METHOD PUBLIC closeAll : BOOL //Return value = TRUE if busy
VAR_INPUT
	Execute													:	BOOL;
END_VAR
	IF Execute
	THEN
		Error												:=	FALSE;
		ErrorId												:= 0;
		SocketCloseAll.bExecute 							:= TRUE;
	ELSIF NOT SocketCloseAll.bBusy  						
	THEN                            						
		Error												:= FALSE;
		ErrorId												:= 0;
		SocketCloseAll.bExecute 							:= FALSE;
	END_IF                          						
                                    	
	MemFnc													:= FNC_CLOSE_ALL;
	THIS^.Execute											:= Execute;

	SocketCloseAll(
		sSrvNetId	:= SrvNetId,
		bExecute	:= ,
		tTimeout	:= Timeout,
		bBusy		=> Busy,
		bError		=> ,
		nErrId		=> );

	IF NOT SocketCloseAll.bBusy
		AND NOT SocketCloseAll.bError
		AND SocketCloseAll.bExecute
	THEN
		Done												:= TRUE;
		MEMSET(ADR(hSocket), 0 , SIZEOF(hSocket));
		hSocketText											:= '';
		Online												:= FALSE;
	ELSE
		Done												:= FALSE;
	END_IF

	IF NOT Busy
	THEN
		IF SocketCloseAll.bExecute
		THEN
			Error											:=	SocketCloseAll.bError;
			IF SocketCloseAll.nErrId >= 16#80070000
			THEN
				ErrorId										:= E_AdsErr.CLIENT_W32ERROR;
				WinsockErrorId								:= ADSERROR_TO_WSERROR(SocketCloseAll.nErrId);
			ELSE                    						
				ErrorId										:= SocketCloseAll.nErrId;
				WinsockErrorId								:= WSOK;
			END_IF
		END_IF
		IF NOT Execute
		THEN
			MemFnc											:=  -1;
			SocketCloseAll(bExecute := FALSE);
		END_IF
	END_IF
	
	CloseAll												:= Busy;
END_METHOD

METHOD PUBLIC connect : BOOL //Return value = TRUE if busy
//required parameter
//Host
//Port
VAR_INPUT
	Execute													:	BOOL;	
END_VAR
	IF Execute
	THEN
		Error												:=	FALSE;
		ErrorId												:= 0;
		SocketCreate.bExecute 								:= TRUE;
	ELSIF NOT SocketCreate.bBusy    						
	THEN                            						
		Error												:=	FALSE;
		ErrorId												:= 0;
		SocketCreate.bExecute 								:= FALSE;
	END_IF                          						
                                    	
	MemFnc													:= FNC_CONNECT;
	THIS^.Execute											:= Execute;

	SocketCreate(
		sSrvNetId	:= SrvNetId,
		sRemoteHost	:= Host,
		nRemotePort	:= Port,
		bExecute	:= ,
		tTimeout	:= Timeout,
		bBusy		=> Busy,
		bError		=> ,
		nErrId		=> ,
		hSocket		=> );

	IF NOT SocketCreate.bBusy
		AND NOT SocketCreate.bError
		AND SocketCreate.bExecute
	THEN
		Done												:= TRUE;
		hSocket												:= SocketCreate.hSocket;
		hSocketText											:= HSOCKET_TO_STRING(hSocket);
		Online												:= SocketCreate.hSocket.handle <> 0;
	ELSE                                					
		Done												:= FALSE;
	END_IF                              	
                                        	
	IF NOT Busy
	THEN
		IF SocketCreate.bExecute
		THEN
			Error											:=	SocketCreate.bError;
			IF SocketCreate.nErrId >= 16#80070000
			THEN
				ErrorId										:= E_AdsErr.CLIENT_W32ERROR;
				WinsockErrorId								:= ADSERROR_TO_WSERROR(SocketCreate.nErrId);
			ELSE                    						
				ErrorId										:= SocketCreate.nErrId;
				WinsockErrorId								:= WSOK;
			END_IF                  						
		END_IF                      	
		IF NOT Execute              	
		THEN
			MemFnc											:= -1;
			SocketCreate(bExecute := FALSE);
		END_IF
	END_IF
	
	Connect													:= Busy;
END_METHOD

METHOD PUBLIC listen : BOOL //Return value = TRUE if busy
//required parameter
//hListener
//Host
//Port
VAR_INPUT
	Execute													:	BOOL;
END_VAR
	IF Execute
	THEN
		Error												:= FALSE;
		ErrorId												:= 0;
		SocketListen.bExecute 								:= TRUE;
	ELSIF NOT SocketListen.bBusy    						
	THEN                            						
		Error												:= FALSE;
		ErrorId												:= 0;
		SocketListen.bExecute 								:= FALSE;
	END_IF                          						
                                        					
	MemFnc													:= FNC_LISTEN;
	THIS^.Execute											:= Execute;
                                        	
	SocketListen(
		sSrvNetId	:= SrvNetId,
		sLocalHost	:= Host,
		nlocalPort	:= Port,
		bExecute	:= ,
		tTimeout	:= Timeout,
		bBusy		=> Busy,
		bError		=>,
		nErrId		=> ,
		hListener	=>	hSocket);

	IF NOT SocketListen.bBusy
		AND NOT SocketListen.bError
		AND SocketListen.bExecute
	THEN
		Done												:= TRUE;
		hSocket												:= SocketListen.hListener;
		hSocketText											:= HSOCKET_TO_STRING(hSocket);
		Request												:= TRUE;
	ELSE                            						
		Done												:= FALSE;
	END_IF                              					
                                        	
	IF NOT Busy
	THEN
		IF SocketListen.bExecute
		THEN
			Error											:=	SocketListen.bError;
			IF SocketListen.nErrId >= 16#80070000
			THEN
				ErrorId										:= E_AdsErr.CLIENT_W32ERROR;
				WinsockErrorId								:= ADSERROR_TO_WSERROR(SocketListen.nErrId);
			ELSE                    						
				ErrorId										:= SocketListen.nErrId;
				WinsockErrorId								:= WSOK;
			END_IF                  						
		END_IF                      	
		IF NOT Execute              	
		THEN                        	
			MemFnc											:= -1;
			SocketListen(bExecute := FALSE);
		END_IF
	END_IF
	
	Listen													:= Busy;
END_METHOD

END_FUNCTION_BLOCK

// POUs/Connectivity/TF6310-TcpServer/UDP/UDPSendRecCtrl
{attribute 'no_check'}
//Send or receive data via TCP connection 
//based on TF6310, required lib: Tc2_TcpIp - see Beckhoff Infosys for more information
FUNCTION_BLOCK UDPSendRecCtrl Extends FbBase
VAR_OUTPUT CONSTANT
	FNC_RECEIVE												:	INT := 0;
	FNC_SEND												:	INT := 1;
END_VAR             										
VAR_INPUT           										
	Fnc														:	INT (FNC_RECEIVE..FNC_SEND) := FNC_RECEIVE;
{attribute 'displaymode':='binary'}
	Options													:	BYTE := 2#0000_0000; // Options Bit .0 = Do NOT restart receive intern / Receive intern nicht neustarten
	SrvNetId												: 	T_AmsNetId := ''; 	// server ams net id
	RemoteHost 												: 	T_IPv4Addr; // Target ip adress - only for send data *)
	RemotePort												: 	UDINT; 	// target port - only for send data *)
	Timeout													: 	TIME := DEFAULT_ADS_TIMEOUT; //ADS timeout
	hSocket													:	T_HSOCKET; 	// Socket handle provided by Server/Handle
	pData													:	POINTER TO BYTE; 	//Pointer do send/res data field 
	cbData													:	UDINT; 	// Size of send/rec data field 
	EnableDebugMode											:	BOOL;	// Write debug information into twincat logger
END_VAR
VAR_OUTPUT
	RecBytes 												:  UDINT;  	// Count of received bytes
	WinsockErrorId											:	E_WinsockError; //Winsocket error enum - see TF6310 documentation for further information
	RecRemoteHost 											:  STRING(15); 	// Remote host IP
	RecRemotePort											:  UDINT; 	// Remote host port
END_VAR                 									
VAR                     	
(* cache ************************************************************)
	MemFnc													:	INT := -1;

(* function-block instances ***************************************************************)
	SocketSend												:	FB_SocketUdpSendTo;
	SocketReceive											:	FB_SocketUdpReceiveFrom;

END_VAR


(* Execute ***************************************************************************************)
	rtExecute(CLK := Execute);
	IF rtExecute.Q
		AND MemFnc < 0
	THEN
		MemFnc 												:= SEL(Fnc = FNC_SEND, FNC_RECEIVE , FNC_SEND) ;
		Busy												:= TRUE;
		Done												:= FALSE;
		Error												:= FALSE;
		ErrorID												:= 0;
	END_IF

(* Call Method ***********************************************************************************)
	CASE MemFnc OF
	FNC_SEND:
		SEND( Execute := Execute);

	FNC_RECEIVE:
		Receive( Execute := Execute);
			
	-1:
		IF NOT Execute
		THEN
			Busy											:= FALSE;
			Done											:= FALSE;
			Error											:= FALSE;
			ErrorID											:= 0;
		END_IF                              				
	ELSE                                    				
		Busy												:= FALSE;
		Done												:= FALSE;
		Error												:= Execute;
		ErrorID												:= E_AdsErr.DEVICE_INVALIDPARM;
	END_CASE                                	
                                            	
(*************************************************************************************************)

PROPERTY PUBLIC optDoNotRestartReceiveCylic : BOOL
GET
optDoNotRestartReceiveCylic := Options.0;
END_GET
SET
Options.0 := optDoNotRestartReceiveCylic;
END_SET
END_PROPERTY

METHOD PUBLIC receive : BOOL	//Return value = TRUE if busy
//required parameter
//hSocket
//pData
//cbData
VAR_INPUT
	Execute													:	BOOL;
END_VAR
	MemFnc													:= FNC_RECEIVE;
	THIS^.Execute											:= Execute;
	
IF pData = 0 
THEN
	Busy													:= NOT Error;
	Error													:= TRUE;
	ErrorId													:= E_AdsErr.DEVICE_INVALIDPARM;
	Done													:= FALSE;
	MemFnc													:= SEL(Execute , -1 ,MemFnc); 
	RETURN;
END_IF

	IF Execute
	THEN
		Error												:=	FALSE;
		ErrorId												:= 0;
		SocketReceive.bExecute 								:= TRUE;
	ELSIF NOT SocketReceive.bBusy       					
	THEN                                					
		Error												:=	FALSE;
		ErrorId												:= 0;
		SocketReceive.bExecute 								:= FALSE;
	END_IF

	SocketReceive(
		sSrvNetId	:= SrvNetId,
		hSocket		:= hSocket,
		cbLen		:= cbData,
		pDest		:= pData,
		bExecute	:= ,
		tTimeout	:= Timeout,
		bBusy		=> Busy,
		bError		=> ,
		nErrId		=> ,
		nRecBytes	=> );

	IF NOT SocketReceive.bBusy
		AND NOT SocketReceive.bError
		AND SocketReceive.bExecute
	THEN
		IF EnableDebugMode
			AND SocketReceive.nRecBytes > 0
			AND NOT Done
		THEN
			hSocket.remoteAddr.sAddr						:= SocketReceive.sRemoteHost;
			hSocket.remoteAddr.nPort						:= SocketReceive.nRemotePort;
			ADSLOGDINT(	ADSLOG_MSGTYPE_ERROR OR ADSLOG_MSGTYPE_LOG, CONCAT('%d Bytes received / ', HSOCKET_TO_STRING(hSocket)) , UDINT_TO_DINT(SocketReceive.nRecBytes));
		END_IF
		Done												:= SocketReceive.nRecBytes > 0 OR Options.0; (* Done melden nach jedenm Lesezyklus, egal ob Daten empfangen wurden *)
		IF NOT Done
		THEN (* Nur Done melden wenn auch was empfangen wurde *)
			SocketReceive(bExecute := FALSE);
			SocketReceive(bExecute := TRUE, bBusy => Busy);
		END_IF
		RecBytes											:= SEL(Done , 0 ,SocketReceive.nRecBytes);
	ELSE                                					
		Done												:= FALSE;
	END_IF                              	

	IF NOT Busy
	THEN
		IF SocketReceive.bExecute
		THEN
			Error											:=	SocketReceive.bError;
			IF SocketReceive.nErrId >= 16#80070000
			THEN
				ErrorId										:= E_AdsErr.CLIENT_W32ERROR;
				WinsockErrorId								:= ADSERROR_TO_WSERROR(SocketReceive.nErrId);
			ELSE                    						
				ErrorId										:= SocketReceive.nErrId;
				WinsockErrorId								:= WSOK;
			END_IF                  						
		END_IF                      	
		IF NOT Execute
		THEN
			MemFnc											:= -1;
			SocketReceive(bExecute := FALSE);
		END_IF
	END_IF
	
	//Method return
	Receive													:= Busy;
END_METHOD

METHOD PUBLIC send : BOOL 	//Return value = TRUE if busy
//required parameter
//hSocket
//pData
//cbData
//RemoteHost
//RemotePort
VAR_INPUT
	Execute													:	BOOL;
END_VAR
	MemFnc													:= FNC_SEND;
	THIS^.Execute											:= Execute;
	                                    					
IF pData = 0 THEN                       					
	Busy													:= NOT Error;
	Error													:= TRUE;
	ErrorId													:= E_AdsErr.DEVICE_INVALIDPARM;
	Done													:= FALSE;
	MemFnc													:= SEL(Execute , -1 ,MemFnc); 
	RETURN;
END_IF

	IF Execute
	THEN
		Error												:= FALSE;
		ErrorId												:= 0;
		SocketSend.bExecute 								:= TRUE;
	ELSIF NOT SocketSend.bBusy          					
	THEN                                					
		Error												:= FALSE;
		ErrorId												:= 0;
		SocketSend.bExecute 								:= FALSE;
	END_IF                              	
	
	SocketSend(
		sSrvNetId	:= SrvNetId,
		hSocket		:= hSocket,
		sRemoteHost	:= RemoteHost,
		nRemotePort	:= RemotePort,
		cbLen		:= cbData,
		pSrc		:= pData,
		bExecute	:= ,
		tTimeout	:= Timeout,
		bBusy		=> Busy,
		bError		=> ,
		nErrId		=> );

	IF NOT SocketSend.bBusy
		AND NOT SocketSend.bError
		AND SocketSend.bExecute
	THEN
		IF NOT Done
			AND EnableDebugMode
		THEN
			hSocket.remoteAddr.sAddr						:= SocketSend.sRemoteHost;
			hSocket.remoteAddr.nPort						:= SocketSend.nRemotePort;
			ADSLOGDINT(	ADSLOG_MSGTYPE_ERROR OR ADSLOG_MSGTYPE_LOG, CONCAT('%d Bytes sended / ', HSOCKET_TO_STRING(hSocket)) , UDINT_TO_DINT(cbData));
		END_IF
		Done												:= TRUE;
	ELSE                                					
		Done												:= FALSE;
	END_IF                              	
                                        	
	IF NOT Busy
	THEN
		IF SocketSend.bExecute
		THEN
			Error											:=	SocketSend.bError;
			IF SocketSend.nErrId >= 16#80070000
			THEN
				ErrorId										:= E_AdsErr.CLIENT_W32ERROR;
				WinsockErrorId								:= ADSERROR_TO_WSERROR(SocketSend.nErrId);
			ELSE                    						
				ErrorId										:= SocketSend.nErrId;
				WinsockErrorId								:= WSOK;
			END_IF                  	
		END_IF
		IF NOT Execute
		THEN
			MemFnc											:= -1;
			SocketSend(bExecute := FALSE);
		END_IF
	END_IF
	
	//Method return
	Send													:= Busy;
END_METHOD

END_FUNCTION_BLOCK

// POUs/Connectivity/TF6310-TcpServer/UDP/UDPServerCtrl
{attribute 'no_check'}
//Helper for UDP Client or Server for socket communications. (Wrapper for Fbs like SocketAccpet,SocketClose,SocketConnect....)
//based on TF6310, required lib: Tc2_TcpIp - see Beckhoff Infosys for more information
FUNCTION_BLOCK UDPServerCtrl 
VAR_INPUT
	Enable													:	BOOL := FALSE;	// FB will be processed as long as enable is TRUE 
	SrvNetId												: 	T_AmsNetId := ''; 	// AmsNet id for TcpIp Server instance - '' for local 
	SrvLocalHost											:	T_IPv4Addr := ''; 	// IP-Adress of local ip-adapter used for server communication
	SrvLocalPort											:	UDINT;			//	IP-Port of local ip-adapter used for server communication

	EnableDebugMode											:	BOOL := FALSE; 	// Write debug information into twincat logger
	CloseAllSocket											:	BOOL := TRUE; 	// Close all socket if server will be diabled - FALSE = close only connected port
END_VAR
VAR_OUTPUT
	hSocket													: 	T_HSOCKET ;	// UDP socket handle
	Online													:	BOOL; 	// Connection is current running 
	State													:	E_SocketConnectionState; //Socket connection state enum
	Busy													:	BOOL;	// Busy is TRUE at the rising edge of Enable and stays TRUE as long as the FB is performing any action. 
	Error													:	BOOL;	// Rising edge of Error informs that an error occurred during the execution of the Function Block #
{attribute 'displaymode':='hex'}
	ErrorId													:	UDINT; 	// Error identification - see ADS return codes and TF6310 documentation at Beckhoff infosys for further information
	WinsockErrorId											:	E_WinsockError; // Winsocket error enum - see TF6310 documentation for further information
END_VAR
VAR
(* function-block instances ***************************************************************)
	SocketCtrl												:	UDPSocketCtrl;

END_VAR


(* Execute ****************************************************)
	SocketCtrl(
		Execute			:= ,
		Fnc				:= ,
		SrvNetId		:= '', (* Server IP *)
		LocalHost		:= SrvLocalHost, (* Own IP *)
		LocalPort		:= SrvLocalPort,
		Timeout			:= t#30s,
		Online			=> Online,
		hSocket			=> hSocket,
		Done			=> ,
		Busy			=> Busy,
		Error			=> Error,
		ErrorId			=> ErrorId,
		WinsockErrorId 	=> WinsockErrorId);

	IF Busy
	THEN
		SocketCtrl.Execute 									:= Enable;
	ELSIF SocketCtrl.Done
	THEN
		IF EnableDebugMode
		THEN
			ADSLOGDINT(	ADSLOG_MSGTYPE_ERROR OR ADSLOG_MSGTYPE_LOG, SocketCtrl.hSocketText, 0);
		END_IF
		SocketCtrl(Execute := FALSE);
		Busy												:= FALSE;
		Error												:= FALSE;
		ErrorId												:= 0;
		WinsockErrorId										:= WSOK;
	ELSIF SocketCtrl.Error
	THEN
		IF NOT Enable
		THEN
			SocketCtrl(Execute := FALSE);
			Busy											:= FALSE;
			Error											:= FALSE;
			ErrorId											:= 0;
			WinsockErrorId									:= WSOK;
		END_IF
	ELSE
		IF Enable
			AND NOT Online
		THEN
			SocketCtrl(Execute := FALSE);
			SocketCtrl.Execute 								:= TRUE;
			SocketCtrl.Fnc 									:= SocketCtrl.FNC_CREATE;
			Busy											:= TRUE;
			Error											:= FALSE;
			ErrorId											:= 0;
			WinsockErrorId									:= WSOK;

		ELSIF Online
			AND NOT Enable
		THEN
			SocketCtrl(Execute := FALSE);
			SocketCtrl.Execute 								:= TRUE;
			SocketCtrl.Fnc 									:= SEL(CloseAllSocket, SocketCtrl.FNC_CLOSE,  SocketCtrl.FNC_CLOSE_ALL);
			Busy											:= TRUE;
			Error											:= FALSE;
			ErrorId											:= 0;
			WinsockErrorId									:= WSOK;
		ELSE
			;
		END_IF
	END_IF

(******************************************************************************)

END_FUNCTION_BLOCK

// POUs/Connectivity/TF6310-TcpServer/UDP/UDPSocketCtrl
{attribute 'no_check'}
//Setup Tcp client or server socket communication 
//based on TF6310, required lib: Tc2_TcpIp - see Beckhoff Infosys for more information
FUNCTION_BLOCK UDPSocketCtrl Extends FbBase
VAR_OUTPUT CONSTANT
 	FNC_CREATE 												:	INT := 0; // Create local socket for UDP communication
 	FNC_CLOSE 												:	INT := 1; // Close specified communication socket
 	FNC_CLOSE_ALL 											:	INT := 2; // Close all communication sockets
END_VAR             										
VAR_INPUT           										
	Fnc														:	INT (FNC_CREATE..FNC_CLOSE_ALL) := FNC_CREATE;
	SrvNetId												: 	T_AmsNetId := ''; (* server ip adress *)
	LocalHost 												: 	T_IPv4Addr := '127.0.0.1'; //local ip adress of requestet network adapter 
	LocalPort												: 	UDINT := 0; // Local communication port
	Timeout													: 	TIME := DEFAULT_ADS_TIMEOUT;
END_VAR             										
VAR_OUTPUT          										
	Online													:	BOOL; (* Connection is running *)
	hSocket													: 	T_HSOCKET; 	// UDP Socket handle
	hSocketText												:	STRING(100); 	// Socket information
	WinsockErrorId											:	E_WinsockError; // Winsocket error enum - see TF6310 documentation for further information
END_VAR
VAR
(* Zwischenspeicher ************************************************************)
	MemFnc													:	INT := -1;
                    										
(* Deklaration Trigger **********************************************************)

(* Zeiten ******************************************************************)

(* Bausteine ***************************************************************)
	SocketCloseAll											:	FB_SocketCloseAll;
	SocketClose												:	FB_SocketClose;
	SocketUdpCreate 										:	FB_SocketUdpCreate;

(* Dummy Speicher **********************************************************)

END_VAR


(* Execute ***************************************************************************************)
	rtExecute(CLK := Execute);
	IF rtExecute.Q
		AND MemFnc < 0
	THEN
		MemFnc 												:= Fnc;
		Busy												:= TRUE;
		Done												:= FALSE;
		Error												:= FALSE;
		ErrorID												:= 0;
	END_IF

(* Call Method ***********************************************************************************)
	CASE MemFnc OF
	FNC_CREATE:
		Create(
			Execute		:= Execute,
			LocalHost	:= LocalHost,
			LocalPort	:= LocalPort);

	FNC_CLOSE:
		Close(Execute := Execute);

	FNC_CLOSE_ALL:
		CloseAll(Execute := Execute);

	-1:
		IF NOT Execute
		THEN
			Busy											:= FALSE;
			Done											:= FALSE;
			Error											:= FALSE;
			ErrorID											:= 0;
		END_IF                              				
	ELSE                                    				
		Busy												:= FALSE;
		Done												:= FALSE;
		Error												:= Execute;
		ErrorID												:= E_AdsErr.DEVICE_INVALIDPARM;
	END_CASE

(*************************************************************************************************)

METHOD PUBLIC close : BOOL //Return value = TRUE if busy
VAR_INPUT
	Execute													:	BOOL;
END_VAR
	IF Execute
	THEN
		Error												:=	FALSE;
		ErrorId												:= 0;
		SocketClose.bExecute 								:= TRUE;
	ELSIF NOT SocketClose.bBusy
	THEN
		Error												:=	FALSE;
		ErrorId												:= 0;
		SocketClose.bExecute 								:= FALSE;
	END_IF

	MemFnc													:= FNC_CLOSE_ALL;
	THIS^.Execute											:= Execute;

	SocketClose(
		sSrvNetId	:= SrvNetId,
		hSocket		:= hSocket,
		bExecute	:= ,
		tTimeout	:= Timeout,
		bBusy		=> Busy,
		bError		=>,
		nErrId		=> );

	IF NOT SocketClose.bBusy
		AND NOT SocketClose.bError
		AND SocketClose.bExecute
	THEN
		Done												:= TRUE;
		hSocketText											:=	CONCAT('UDP Socket Close:', HSOCKET_TO_STRING(hSocket));
		hSocketText											:= '';
		Online												:= FALSE;
	ELSE                                					
		Done												:= FALSE;
	END_IF

	IF NOT Busy
	THEN
		IF SocketClose.bExecute
		THEN
			Error											:=	SocketClose.bError;
			IF SocketClose.nErrId >= 16#80070000
			THEN
				ErrorId										:= E_AdsErr.CLIENT_W32ERROR;
				WinsockErrorId								:= ADSERROR_TO_WSERROR(SocketClose.nErrId);
			ELSE                    						
				ErrorId										:= SocketClose.nErrId;
				WinsockErrorId								:= WSOK;
			END_IF
		END_IF
		IF NOT Execute
		THEN
			MemFnc											:= -1;
			SocketClose(bExecute := FALSE);
		END_IF
	END_IF
	
	Close													:= Busy;
END_METHOD

METHOD PUBLIC closeAll : BOOL //Return value = TRUE if busy
VAR_INPUT
	Execute													:	BOOL;
END_VAR
	IF Execute
	THEN
		Error												:=	FALSE;
		ErrorId												:= 0;
		SocketCloseAll.bExecute 							:= TRUE;
	ELSIF NOT SocketCloseAll.bBusy      					
	THEN                                					
		Error												:=	FALSE;
		ErrorId												:= 0;
		SocketCloseAll.bExecute 							:= FALSE;
	END_IF                          						
                                    						
	MemFnc													:= FNC_CLOSE_ALL;
	THIS^.Execute											:= Execute;

	SocketCloseAll(
		sSrvNetId	:= SrvNetId,
		bExecute	:= ,
		tTimeout	:= Timeout,
		bBusy		=> Busy,
		bError		=> ,
		nErrId		=> );

	IF NOT SocketCloseAll.bBusy
		AND NOT SocketCloseAll.bError
		AND SocketCloseAll.bExecute
	THEN
		Done												:= TRUE;
		hSocketText											:= 'UDP Socket Close All';
		Online												:= FALSE;
	ELSE                                					
		Done												:= FALSE;
	END_IF

	IF NOT Busy
	THEN
		IF SocketCloseAll.bExecute
		THEN
			Error											:=	SocketCloseAll.bError;
			IF SocketCloseAll.nErrId >= 16#80070000
			THEN
				ErrorId										:= E_AdsErr.CLIENT_W32ERROR;
				WinsockErrorId								:= ADSERROR_TO_WSERROR(SocketCloseAll.nErrId);
			ELSE                    						
				ErrorId										:= SocketCloseAll.nErrId;
				WinsockErrorId								:= WSOK;
			END_IF
		END_IF
		IF NOT Execute
		THEN
			MemFnc											:= -1;
			SocketCloseAll(bExecute := FALSE);
		END_IF
	END_IF
	
	CloseAll												:= Busy;
END_METHOD

METHOD PUBLIC create : BOOL //Return value = TRUE if busy
//required parameter
//LocalHost
//LocalPort
VAR_INPUT
	Execute													:	BOOL;
	LocalHost 												: 	T_IPv4Addr; (* Own ip adress form requestet Networkadapter *)
	LocalPort												: 	UDINT;
END_VAR
	IF Execute
	THEN
		Error												:=	FALSE;
		ErrorId												:= 0;
		SocketUdpCreate.bExecute 							:= TRUE;
	ELSIF NOT SocketUdpCreate.bBusy     					
	THEN                                					
		Error												:=	FALSE;
		ErrorId												:= 0;
		SocketUdpCreate.bExecute 							:= FALSE;
	END_IF                              					
                                        	
	MemFnc													:= FNC_CREATE;
	THIS^.Execute											:= Execute;
	
	SocketUdpCreate(
		sSrvNetId	:= SrvNetId,
		sLocalHost	:= LocalHost,
		nLocalPort	:= LocalPort,
		bExecute	:= ,
		tTimeout	:= Timeout,
		bBusy		=> Busy,
		bError		=> ,
		nErrId		=> ,
		hSocket		=> );

	IF NOT SocketUdpCreate.bBusy
		AND NOT SocketUdpCreate.bError
		AND SocketUdpCreate.bExecute
	THEN
		Done												:= TRUE;
		hSocket												:= SocketUdpCreate.hSocket;
		Online												:= SocketUdpCreate.hSocket.handle <> 0;
		hSocketText											:=	CONCAT('UDP Socket Create:', HSOCKET_TO_STRING(hSocket));
	ELSE                                					
		Done												:= FALSE;
	END_IF                              	
                                        	
	IF NOT Busy                         	
	THEN
		IF SocketUdpCreate.bExecute
		THEN
			Error											:=	SocketUdpCreate.bError;
			IF SocketUdpCreate.nErrId >= 16#80070000
			THEN
				ErrorId										:= E_AdsErr.CLIENT_W32ERROR;
				WinsockErrorId								:= ADSERROR_TO_WSERROR(SocketUdpCreate.nErrId);
			ELSE                    						
				ErrorId										:= SocketUdpCreate.nErrId;
				WinsockErrorId								:= WSOK;
			END_IF                  	
		END_IF
		IF NOT Execute
		THEN
			MemFnc											:= -1;
			SocketUdpCreate(bExecute := FALSE);
		END_IF
	END_IF
	
	Create													:= Busy;
END_METHOD

END_FUNCTION_BLOCK

// POUs/Connectivity/TF6340-SerialCom/ComPortBackground
{attribute 'no_check'}
//Wrapper for background communication of serial com ports like EL terminal or PC-COM-Port
//based on TF6340 - SerialCommunication (Tc2_SerialCom)
FUNCTION_BLOCK ComPortBackground
VAR_INPUT
	Enable													: BOOL ; // FB will be processed as long as enable is TRUE 
	ResetTrig												: BOOL ; // The function block will be reset with a rising edge 
	Mode													: ComSerialLineMode_t := SERIALLINEMODE_EL6_22B; //terminal parameter, see ComSerialLineMode_t at documentation of library
	pComIn													: POINTER TO BYTE;	// COM-Port process image	%I*
	pComOut													: POINTER TO BYTE;	// COM-Port process image  	%Q* 
	SizeComIn												: UINT := 22; 	// Size of process data - depends on terminal type (3,5,22,64 Byte)
	Cfg 													: ComSerialConfig := (Baudrate := 19200); // Cfg Structure for PC-com port
	TXBuffer												: COMbuffer ;	// TX buffer used by ComPortSendRec
END_VAR
VAR_OUTPUT
	RXBuffer												: COMbuffer ;	// RX buffer used by ComPortSendRec
	PortOpened												: BOOL;	// Background communication etablished
	Busy													: BOOL;	// Busy is TRUE at the rising edge of Enable and stays TRUE as long as the FB is performing any action. 
	Error													: BOOL; // Rising edge of Error informs that an error occurred during the execution of the Function Block 
{attribute 'displaymode':='hex'}
	ErrorId													: UDINT;// Error identification - see ADS return codes and TF6340 documentation at Beckhoff infosys for further information
	ComErrorId												: ComError_t ; 	// Serial com. error indentification - Tc2_SerialCom documentaion for further information
END_VAR
VAR_IN_OUT
END_VAR
VAR
(* internally used variables ********************************************************)
	MemErrorID												: UDINT := 0;
	state													: INT := 0;
	
(* internal function-block instances for serial communication ***************************************************************)
	_ClearComBuffer											: 	ClearComBuffer; // clears the internal communication buffer of the PLC
	_SerLineControl											: 	SerialLineControl; // looks after backround-communication
	_SerLineControlADS										: 	SerialLineControlADS; // looks after backround-communication
	_Comreset												: 	ComReset; // Reset KL-Terminal

END_VAR

(*******************************************************************************)

CASE state OF
0:
	IF NOT Enable AND NOT _SerLineControlADS.Busy
		OR Error
	THEN
		Busy												:= FALSE;
		PortOpened											:= FALSE;
		
		IF ResetTrig
		THEN
			reset();
		END_IF

	ELSIF Mode = ComSerialLineMode_t.SERIALLINEMODE_PC_COM_PORT
	THEN
		_SerLineControlADS(	Connect		:= Enable,
							SerialCfg	:= Cfg,
							NetId		:= '',
							Timeout		:= ,
							TxBuffer	:= TXBuffer,
							RxBuffer	:= RXBuffer,
							PortOpened	=> PortOpened,
							Error		=> ,
							ErrorID		=> ,
							Busy		=> ,
							TxBufCount	=> ,
							RxBufCount	=> );
		
		Busy 												:= TRUE;

		IF _SerLineControlADS.Error 
		THEN
			Error											:= TRUE;
			ErrorId											:= _SerLineControlAds.ErrorId;
//			ComErrorId										:= _SerLineControlAds.ErrorId; // missing cast !
		END_IF

	ELSIF Enable
	THEN
		_SerLineControl(
			Mode		:= mode ,
			pComIn		:= pComIn ,
			pComOut		:= pComOut ,
			SizeComIn	:= UINT_TO_INT(SizeComIn),
			TxBuffer	:= TXBuffer ,
			RxBuffer	:= RXBuffer ,
			Error		=> ,
			ErrorID		=> );
		
		Busy												:= TRUE;

		IF _SerLineControl.Error 
		THEN
			Error											:= TRUE;
			ErrorId											:= TO_UDINT(_SerLineControl.ErrorId);
			ComErrorId										:= _SerLineControl.ErrorId;
		ELSE
			PortOpened										:= TRUE;
		END_IF
	END_IF

20: (* Reset ******************************************)
	_ComReset(	Execute		:= FALSE,
				pComIn		:= pComIn,
				pComOut		:= pComOut ,
				SizeComIn	:= SizeComIn ,
				Done		=> ,
				Busy		=> ,
				Error		=> ,
				ErrorID		=> );

	(* Buffer leeren *)
	_ClearComBuffer(Buffer:= TXBuffer);
	_ClearComBuffer(Buffer:= RXBuffer);

	state 													:= 21;

21:
	_ComReset(	Execute		:= Mode <> ComSerialLineMode_t.SERIALLINEMODE_PC_COM_PORT,
				pComIn		:= pComIn,
				pComOut		:= pComOut ,
				SizeComIn	:= SizeComIn ,
				Done		=> ,
				Busy		=> ,
				Error		=> ,
				ErrorID		=> );
										
	IF NOT _ComReset.Busy
	THEN
		IF _ComReset.Error
		THEN
			Error											:= TRUE;
			ErrorId											:= INT_TO_UDINT(_ComReset.ErrorID);
			ComErrorId										:= _ComReset.ErrorID;
		END_IF
		_ComReset(Execute := FALSE, pComIn	:= pComIn, pComOut := pComOut , SizeComIn := SizeComIn);
		State 												:= SEL(Mode = ComSerialLineMode_t.SERIALLINEMODE_PC_COM_PORT, 0, 90);
	END_IF

90: (* Error ******************************************)
	_SerLineControlADS(	Connect		:= FALSE,
						SerialCfg	:= Cfg,
						NetId		:= '',
						Timeout		:= ,
						TxBuffer	:= TXBuffer,
						RxBuffer	:= RXBuffer,
						PortOpened	=> PortOpened,
						Error		=> ,
						ErrorID		=> ,
						Busy		=> ,
						TxBufCount	=> ,
						RxBufCount	=> );

	IF NOT _SerLineControlADS.Busy
	THEN
		PortOpened											:= FALSE;
		Busy												:= FALSE;
		state												:= 0;
	END_IF
	
END_CASE


(***********************************************************************************************)

METHOD PUBLIC reset : BOOL //Return value = TRUE if execution finished
VAR_INPUT
END_VAR
IF Error OR NOT Enable
THEN //jump to reset state
	state 													:= SEL(state < 20 OR state > 21 ,state , 20);
	Error													:= FALSE;
	ErrorId													:= 0;
	ComErrorId												:= ComError_t.COMERROR_NOERROR;
END_IF
reset													:= TRUE;
END_METHOD

END_FUNCTION_BLOCK

// POUs/Connectivity/TF6340-SerialCom/ComPortSendRec
{attribute 'no_check'}
//Discription: "ComPortSendRecCtrl" can be used to send and receive data and strings via serial Com-Port
//based on TF6340 - SerialCommunication (Tc2_SerialCom)
FUNCTION_BLOCK ComPortSendRec
VAR_OUTPUT CONSTANT
	FNC_RECEIVE												: INT := 0;
	FNC_SEND												: INT := 1;
	
{attribute 'displaymode':='binary'}
	OPTION_STRING_MODE										: BYTE := 2#0000_0001; // Activate String Mode / FALSE = Data mode
{attribute 'displaymode':='binary'}
	OPTION_CLEAR_BUFFER										: BYTE := 2#0000_0010; // Clear ComBuffer/Resetting at with first flag of execute 	
{attribute 'displaymode':='binary'}
	OPTION_REMOVE_PREFIX									: BYTE := 2#00000100; // Remonves Prefix of Received String
{attribute 'displaymode':='binary'}
	OPTION_REMOVE_SUFFIX									: BYTE := 2#00001000; // Remonves Suffix of Received String 	
END_VAR
VAR_INPUT
	Execute													: BOOL := FALSE; 	// The function block will be executed with a rising edge 
	Fnc														: INT (FNC_RECEIVE..FNC_SEND) := FNC_RECEIVE; //
{attribute 'displaymode':='binary'}
	Options													: BYTE := OPTION_STRING_MODE OR OPTION_CLEAR_BUFFER; // Bit 0 = Mode String / Bit 1 = Clear ComBuffer/Resetting at with first flag of execute 	
	Prefix 													: STRING(20) := ''; // e.g. $02 Start of Text 
	Suffix 													: STRING(20) := ''; // e.g. $03 End of Text
	Timeout													: TIME := DEFAULT_ADS_TIMEOUT; //ADS timeout
	SendString												: STRING(MAX_STRING_LENGTH);
	LenghtData												: UDINT; // contains the number, in bytes, of the data to be read
	pSendData												: POINTER TO BYTE := 0; // Pointer at startadress of send data
	pRecData												: POINTER TO BYTE := 0; // Pointer at startadress of receive data
	pRXBuffer												: POINTER TO COMbuffer := 0; // Pointer at RX-Buffer
	pTXBuffer												: POINTER TO COMbuffer := 0; // Pointer at TX-Buffer
END_VAR
VAR_IN_OUT
END_VAR
VAR_OUTPUT
	RecString												: STRING(MAX_STRING_LENGTH); // Received string in case Options bit .0 is set to TRUE
	LenRecData												: INT;	//Len or size of received data
	Busy													: BOOL := FALSE; // Busy is TRUE at the rising edge of Execute and FALSE when one of the outputs Done, Aborted, or Error is set 
	Done													: BOOL := FALSE; // The Done output is set when the commanded action has been completed successfully 
	Error													: BOOL := FALSE; // Error identification - see ADS return codes and TF6340 documentation at Beckhoff infosys for further information
	ComErrorId												: Tc2_SerialCom.ComError_t := COMERROR_NOERROR; // Serial com. error indentification - Tc2_SerialCom documentaion for further information
END_VAR
VAR
(* Local variables **************************************************)
	StateRec												: INT := 0;
	StateSend												: INT := 0;
	MemErrorId												: Tc2_SerialCom.ComError_t := COMERROR_NOERROR; // see also ComLibV2.Lib 
	MemFnc													: INT := -1;
	
	RecDataPrefixArr										: ARRAY[1..20] OF BYTE;
	RecDataSuffixArr										: ARRAY[1..20] OF BYTE;

(* Trigger **********************************************************)
	RT_Execute												: R_Trig;
	
(* Instances ***************************************************************)
	_ClearComBuffer											: Tc2_SerialCom.ClearComBuffer ;	
	_RecString												: Tc2_SerialCom.ReceiveString255 ;
	_SendString												: Tc2_SerialCom.SendString255 ;
	_SendData												: Tc2_SerialCom.SendData;
	_RecData												: Tc2_SerialCom.ReceiveData;	
END_VAR

(* Execute ***************************************************************************************)
	RT_Execute(CLK := Execute);
	IF RT_Execute.Q
		AND MemFnc < 0
	THEN
		MemFnc 												:= Fnc;
		Busy												:= TRUE;
		Done												:= FALSE;
		Error												:= FALSE;
		ComErrorId											:= COMERROR_NOERROR; 
	END_IF                                 				
                                            	
(* Call Method ***********************************************************************************)
	CASE MemFnc OF
	FNC_RECEIVE:
		IF Options.0
		THEN //Str mode 
			ReceiveStr(Execute:= Execute);
		ELSE //Data mode
			ReceiveData(Execute:= Execute);
		END_IF
	
	FNC_SEND:
		IF Options.0
		THEN //Str mode 
			SendStr(Execute:= Execute);
		ELSE //Data mode
			SendData(Execute:= Execute);
		END_IF	
		
	-1:
		IF NOT Execute
		THEN
			Busy											:= FALSE;
			Done											:= FALSE;
			Error											:= FALSE;
			ComErrorId										:= COMERROR_NOERROR; 
		END_IF                              				
	ELSE                                    				
		Busy												:= FALSE;
		Done												:= FALSE;
		Error												:= Execute;
		ComErrorId											:= COMERROR_PARAMETERCHANGED; 
	END_CASE                                	
                                            	
(*************************************************************************************************)

METHOD PUBLIC clearBuffer : booL //Return value = TRUE if execution finished
//required parameter
//pTXBuffer
//pRXBuffer
VAR_INPUT
END_VAR
reset();

IF 	pRXBuffer = 0 OR pTXBuffer = 0
THEN
	Busy													:= FALSE;
	Done													:= FALSE;
	Error 													:= TRUE;
	ComErrorId 												:= COMERROR_INVALIDPOINTER;
ELSE                        								
	_ClearComBuffer(Buffer:= pTXBuffer^);
	_ClearComBuffer(Buffer:= pRXBuffer^);
	
END_IF
ClearBuffer													:= TRUE;
END_METHOD

PROPERTY PUBLIC optClearBuffer : BOOL
GET
optClearBuffer := Options.1;
END_GET
SET
Options.1 := optClearBuffer;
END_SET
END_PROPERTY

{attribute 'monitoring' := 'call'}
PROPERTY PUBLIC optEnableStringMode : BOOL
GET
optEnableStringMode := Options.0;
END_GET
SET
Options.0 := optEnableStringMode;
END_SET
END_PROPERTY

PROPERTY PUBLIC optRemovePrefix : BOOL
GET
optRemovePrefix := Options.2;
END_GET
SET
Options.2 := optRemovePrefix;
END_SET
END_PROPERTY

PROPERTY PUBLIC optRemoveSuffix : BOOL
GET
optRemoveSuffix := Options.3;
END_GET
SET
Options.3 := optRemoveSuffix;
END_SET
END_PROPERTY

METHOD PUBLIC receiveData : BOOL //Return value = TRUE if busy
//required parameter
//pRXBuffer
//pRecData
//LenghtData
//Prefix
//Suffix
VAR_INPUT
	Execute													:	BOOL; 
END_VAR
IF 	pRXBuffer = 0 OR pRecData = 0 
THEN
	Busy													:= NOT Error;
	Error													:= TRUE;
	ComErrorId 												:= COMERROR_INVALIDPOINTER;
	Done													:= FALSE;
	MemFnc													:= -1 ;
	RETURN;
END_IF

IF 	Execute
	AND StateRec = 0
THEN 
	IF Options.1
	THEN
		reset();
		_ClearComBuffer(Buffer:= pRXBuffer^);
	END_IF
	StateRec												:= 1;		
END_IF

MemFnc														:= FNC_RECEIVE;

THIS^.Execute												:= Execute;

IF StateRec = 1
THEN
	_RecData.LenPrefix 										:= UDINT_TO_BYTE(HEXSTR_TO_DATA(Prefix,ADR(RecDataPrefixArr), SIZEOF(RecDataPrefixArr)));
	_RecData.LenSuffix 										:= UDINT_TO_BYTE(HEXSTR_TO_DATA(Suffix,ADR(RecDataSuffixArr), SIZEOF(RecDataSuffixArr)));

// receiving data
	_RecData(
		pPrefix			:= ADR(RecDataPrefixArr),
		LenPrefix		:= , // see above
		pSuffix			:= ADR(RecDataSuffixArr),
		LenSuffix		:= , // see above
		pReceiveData	:= pRecData,
		SizeReceiveData	:= LenghtData,
		Timeout			:= Timeout,
		Reset			:= FALSE,
		RXbuffer		:= pRXBuffer^,
		DataReceived	=> ,
		busy			=> ,
		Error			=> ,
		RxTimeout		=> ,
		LenReceiveData	=> );
		
	IF _RecData.Error <> 0
	THEN
		StateRec											:= 90;
	ELSIF NOT _RecData.Busy
		AND _RecData.DataReceived
	THEN
		StateRec											:= 2;
		LenRecData											:= TO_INT(_RecData.LenReceiveData);
	ELSIF NOT _RecData.Busy
		AND _RecData.RxTimeout
	THEN
		StateRec											:= 91;
	ELSE
		LenRecData											:= TO_INT(_RecData.LenReceiveData);
	END_IF
END_IF

CASE stateRec OF
0: ; //waiting til start
	ComErrorId												:= COMERROR_NOERROR; 
	Busy													:= FALSE;
	Error													:= FALSE;
	Done													:= FALSE;
	
1: ; //reading acticve
	ComErrorId												:= COMERROR_NOERROR; 
	Busy													:= TRUE;
	Error													:= FALSE;
	Done													:= FALSE;
	
2: // finished reading
	ComErrorId												:= COMERROR_NOERROR; 
	Busy													:= FALSE;
	Error													:= FALSE;
	Done													:= TRUE;
	
	IF NOT Execute		
	THEN
		MemFnc												:= -1;
		StateRec											:= 0;
	END_IF
	
90:
	ComErrorId												:= _RecData.Error; 
	MemErrorId												:= ComErrorId;
	Busy													:= FALSE;
	Error													:= TRUE;
	Done													:= FALSE;
	
	IF NOT Execute		
	THEN
		MemFnc												:= -1;
		StateRec											:= 0;
	END_IF
	
91:	
	ComErrorId												:= COMERROR_TIMEOUT; 
	MemErrorId												:= ComErrorId;
	Busy													:= FALSE;
	Error													:= TRUE;
	Done													:= FALSE;
	
	IF NOT Execute		
	THEN
		MemFnc												:= -1;
		StateRec											:= 0;
	END_IF
END_CASE

ReceiveData													:= Busy;
END_METHOD

METHOD PUBLIC receiveStr : BOOL //Return value = TRUE if busy
//required parameter
//pRXBuffer
//Prefix
//Suffix
VAR_INPUT
	Execute													:	BOOL;
END_VAR
IF pRXBuffer = 0 THEN
	Busy													:= NOT Error;
	Error													:= TRUE;
	ComErrorId												:= COMERROR_INVALIDPOINTER;
	Done													:= FALSE;
	MemFnc													:= -1 ;
	RETURN;
END_IF

IF Execute
	AND StateRec = 0
THEN //start reading
	IF Options.1
	THEN
		reset();
		_ClearComBuffer(Buffer:= pRXBuffer^);	
	END_IF
	StateRec												:= 1;
	MemSet(ADR(RecString),0,SIZEOF(RecString));						
END_IF

MemFnc														:= FNC_RECEIVE;

THIS^.Execute												:= Execute;

IF StateRec = 1
THEN
	_RecString(
		Prefix			:= Prefix ,
		Suffix			:= Suffix ,
		Timeout			:= Timeout ,
		Reset			:= FALSE,
		ReceivedString	:= RecString,
		RXbuffer		:= pRXBuffer^,
		StringReceived	=> ,
		Busy			=> ,
		Error			=> ,
		RxTimeout		=> );
		
	IF _RecString.Error <> 0
	THEN
		StateRec											:= 90;
	ELSIF NOT _RecString.Busy
		AND _RecString.StringReceived
	THEN
		IF Options.2 THEN RecString 						:= DELETE(RecString, len(Prefix), 1); 				END_IF
		IF Options.3 THEN RecString 						:= DELETE(RecString, len(Suffix), len(RecString)); 	END_IF
		LenRecData											:= LEN(RecString);
		StateRec											:= 2;

	ELSIF NOT _RecString.Busy
		AND _RecString.RxTimeout
	THEN
		StateRec											:= 91;
	END_IF
END_IF

CASE stateRec OF
0: ; //wait until start
	ComErrorId												:= COMERROR_NOERROR; 
	Busy													:= FALSE;
	Error													:= FALSE;
	Done													:= FALSE;
	                        								
1: ; //reading active       								
	ComErrorId												:= COMERROR_NOERROR; 
	Busy													:= TRUE;
	Error													:= FALSE;
	Done													:= FALSE;
	                        								
2: // reading finished      								
	ComErrorId												:= COMERROR_NOERROR; 
	Busy													:= FALSE;
	Error													:= FALSE;
	Done													:= TRUE;
	IF NOT Execute		    								
	THEN                    								
		MemFnc												:= -1;
		StateRec											:= 0;
	END_IF                  								
	                        								
90:                         								
	ComErrorId												:= _RecString.Error; 
	MemErrorId												:= ComErrorId;
	Busy													:= FALSE;
	Error													:= TRUE;
	Done													:= FALSE;
	IF NOT Execute		    								
	THEN                    								
		MemFnc												:= -1;
		StateRec											:= 0;
	END_IF                  								
	                        								
91:                         								
	ComErrorId												:= COMERROR_TIMEOUT; 
	MemErrorId												:= ComErrorId;
	Busy													:= FALSE;
	Error													:= TRUE;
	Done													:= FALSE;
	IF NOT Execute		    								
	THEN                    								
		MemFnc												:= -1;
		StateRec											:= 0;
	END_IF                  								
END_CASE                    								
                            								
ReceiveStr													:= Busy;
END_METHOD

METHOD PUBLIC reset : bool //Return value = TRUE if execution finished
//required parameter
//pRXBuffer
VAR_INPUT
END_VAR
IF pRXBuffer = 0 
THEN
	Busy													:= NOT Error;
	Error													:= TRUE;
	ComErrorId 												:= COMERROR_INVALIDPOINTER;
	Done													:= FALSE;
	MemFnc													:= -1 ;
	reset													:= TRUE;
	RETURN;                             					
END_IF                                  					
                                        					
	Busy													:= FALSE;
	Done													:= FALSE;
	Error													:= FALSE;
	ComErrorId												:= COMERROR_NOERROR; // see also ComLibV2.Lib
	StateRec												:= 0;
	StateSend												:= 0;
                                        					
	_RecString(                             				
		Prefix			:= Prefix ,
		Suffix			:= Suffix ,
		Timeout			:= Timeout ,
		Reset			:= TRUE,
		ReceivedString	:= RecString,
		RXbuffer		:= pRXBuffer^,
		StringReceived	=> ,
		Busy			=> ,
		Error			=> ,
		RxTimeout		=> );
		
	_RecString.Reset										:= FALSE;

	_RecData(
		pPrefix			:= ADR(RecDataPrefixArr),
		LenPrefix		:= , // see above
		pSuffix			:= ADR(RecDataSuffixArr),
		LenSuffix		:= , // see above
		pReceiveData	:= pRecData,
		SizeReceiveData	:= LenghtData,
		Timeout			:= Timeout,
		Reset			:= TRUE,
		RXbuffer		:= pRXBuffer^,
		DataReceived	=> ,
		busy			=> ,
		Error			=> ,
		RxTimeout		=> ,
		LenReceiveData	=> );
	_RecData.Reset											:= FALSE;		
		
	reset													:= TRUE;
END_METHOD

METHOD PUBLIC sendData : BOOL //Return value = TRUE if busy
//required parameter
//pTXBuffer
//pSendData
//LenghtData		
VAR_INPUT
	Execute													:	BOOL;
END_VAR
IF 	pTXBuffer = 0 
	OR pSendData = 0 
THEN
	Busy													:= NOT Error;
	Error													:= TRUE;
	ComErrorId 												:= COMERROR_INVALIDPOINTER;
	Done													:= FALSE;
	MemFnc													:= -1 ;
	RETURN;                             					
END_IF

	IF Execute
		AND StateSend = 0
	THEN // start reading
		IF Options.1
		THEN
			reset();
			_ClearComBuffer(Buffer:= pTXBuffer^);
		END_IF
		StateSend											:= 1;		
	END_IF

	MemFnc													:= FNC_SEND;
	
	THIS^.Execute											:= Execute;
		
	IF 	StateSend = 1 
		OR StateSend = 2
	THEN		
		_SendData(
			pSendData 	:= pSendData,
			Length		:= LenghtData,
			TXbuffer	:= pTXBuffer^,
			Busy		=> ,
			Error		=> );
			
		IF StateSend = 1
		THEN
			StateSend 		:= 2;
		ELSIF _SendData.Error <> 0
		THEN
			StateSend		:= 90;
		ELSIF NOT _SendData.Busy
		THEN
			StateSend		:= 3;
		END_IF
	END_IF
	
	CASE StateSend OF
	0: ; //wait until start
		ComErrorId											:= COMERROR_NOERROR; 
		Busy												:= FALSE;
		Error												:= FALSE;
		Done												:= FALSE;
		                        							
	1,2: ; //writing active     							
		ComErrorId											:= COMERROR_NOERROR; 
		Busy												:= TRUE;
		Error												:= FALSE;
		Done												:= FALSE;
		                        							
	3: // finished writing      							
		ComErrorId											:= COMERROR_NOERROR; 
		Busy												:= FALSE;
		Error												:= FALSE;
		Done												:= TRUE;
		IF NOT Execute		    							
		THEN                    							
			MemFnc											:= -1;
			StateSend										:= 0;
		END_IF                  							
		                        							
	90:                         							
		ComErrorId											:= _SendData.Error; 
		MemErrorId											:= ComErrorId;
		Busy												:= FALSE;
		Error												:= TRUE;
		Done												:= FALSE;
		IF NOT Execute		    							
		THEN                    							
			MemFnc											:= -1;
			StateSend										:= 0;
		END_IF                  							
		                        							
	END_CASE                    							
	                            							
	SendData												:= Busy;
END_METHOD

METHOD PUBLIC sendStr : BOOL //Return value = TRUE if busy
//required parameter
//pTXBuffer
//SendString
VAR_INPUT
	Execute													:	BOOL;
END_VAR
IF pTXBuffer = 0 THEN
	Busy													:= NOT Error;
	Error													:= TRUE;
	ComErrorId 												:= COMERROR_INVALIDPOINTER;
	Done													:= FALSE;
	MemFnc													:= -1 ;
	RETURN;
END_IF

IF 	Execute
	AND StateSend = 0
THEN //start reading
	IF Options.1
	THEN
		reset();
		_ClearComBuffer(Buffer:= pTXBuffer^);
	END_IF
	StateSend												:= 1;		
END_IF                                              	
                                                    	
MemFnc														:= FNC_SEND;
                                                    	
THIS^.Execute												:= Execute;
                                                    	
IF 	StateSend = 1                                   	
	OR StateSend = 2                                	
THEN		                                        	
	_SendString(                                    	
		SendString	:= SendString,                  	
		TXbuffer	:= pTXBuffer^,                  	
		Busy		=> ,                            	
		Error		=> );                           	
					                                	
	IF StateSend = 1                                	
	THEN                                            	
		StateSend											:= 2;
	ELSIF _SendData.Error <> 0                      	
	THEN                                            	
		StateSend											:= 90;
	ELSIF NOT _SendData.Busy                        	
	THEN                                            	
		StateSend											:= 3;
	END_IF                                          	
END_IF                                              	
                                                    	
CASE StateSend OF                                   	
0: ; //wait until start                             	
	ComErrorId												:= COMERROR_NOERROR;    	
	Busy													:= FALSE;               	
	Error													:= FALSE;               	
	Done													:= FALSE;               	
	                        								                        	
1,2: ; //writing active     								                        	
	ComErrorId												:= COMERROR_NOERROR;    	
	Busy													:= TRUE;                	
	Error													:= FALSE;               	
	Done													:= FALSE;               	
	                        								                        	
3: // finished writing      								                        	
	ComErrorId												:= COMERROR_NOERROR;    	
	Busy													:= FALSE;               	
	Error													:= FALSE;               	
	Done													:= TRUE;                	
	IF NOT Execute		    								                        	
	THEN                    								                        	
		MemFnc												:= -1;                  	
		StateSend											:= 0;                   	
	END_IF                  								                        	
	                        								                        	
90:                         								                        	
	ComErrorId												:= _SendString.Error;   	
	MemErrorId												:= ComErrorId;          	
	Busy													:= FALSE;               	
	Error													:= TRUE;                	
	Done													:= FALSE;               	
	IF NOT Execute		    								                        	
	THEN                    								                        	
		MemFnc												:= -1;                  	
		StateSend											:= 0;                   	
	END_IF                  								                        	
	                        								                        	
END_CASE                    								                        	
                            								                        	
SendStr														:= Busy;
END_METHOD

END_FUNCTION_BLOCK

// POUs/Connectivity/isValidIPv4Addr
//Checks wheter a IPv4 address string is valid
FUNCTION isValidIPv4Addr : bool
VAR_INPUT
	IPv4Addr				:	T_IPv4Addr; //String
END_VAR
VAR
	Bytes 					: 	T_IPv4AddrArr; //IPv4 address as an array 0..3 of Byte
END_VAR

Bytes						:= F_ScanIPv4AddrIds(IPv4Addr);
isValidIPv4Addr				:= Bytes[0] > 0 AND Bytes[0] <= 255
								AND Bytes[1] >= 0 AND Bytes[1] <= 255
								AND Bytes[2] >= 0 AND Bytes[2] <= 255
								AND Bytes[3] >= 0 AND Bytes[3] <= 255;

END_FUNCTION

// POUs/ControllerTools/AverageFilter
//LREAL average filter
FUNCTION_BLOCK AverageFilter
VAR_INPUT	
	IN														: LREAL;		// Adds value for average calculation
END_VAR
VAR_OUTPUT
	Q														: LREAL:=0.0;	// Result of average calculation
	Valid													: BOOL:=FALSE;	// Is TRUE once a value is inserted
END_VAR         											
VAR             											
	Total													: LREAL:=0.0;
	Count													: LREAL:=0;
END_VAR

Insert(IN);

METHOD PUBLIC clear : booL; //Return value = TRUE if execution finished
VAR_INPUT
END_VAR
Q:=Total	:=0.0;
Valid		:=FALSE;
Count		:=0.0;
Clear		:= TRUE;
END_METHOD

METHOD PUBLIC insert : LREAL //Result = actual average value
VAR_INPUT
	Value								:	LREAL ;
END_VAR
Total		:=Total+Value;
Count		:=Count+1.0;
Q			:=Total/Count;
Valid		:=TRUE;
Insert 		:= Q;
END_METHOD

END_FUNCTION_BLOCK

// POUs/ControllerTools/PIDController
//Base PID controller with manual 
FUNCTION_BLOCK PIDController 
VAR_INPUT
	Enable													: BOOL := FALSE;	// FB will be processed as long as enable is TRUE 
	ResetTrig												: BOOL := FALSE;	// The function block will get reseted with a rising edge 
	ManualOn												: BOOL := FALSE;	// set Q to ManualValue 
	Sync													: BOOL := FALSE;	// synchronization flag for bumpless initialisation
	// controller input (deviation)   					
	SetValue												: LREAL := 0.0;		// Setpoint value										
	ActValue												: LREAL := 0.0;		// Actual value											
	
	MinOutput												: LREAL := 0.0;		// controller minimum output (min. limit)				
	MaxOutput												: LREAL := 0.0;		// controller maximum output (max. limit)				
	SyncValue												: LREAL := 0.0;		// syncronization value for bumpless init.				
	ManualValue												: LREAL := 0.0;		// manual value *)
	// controller values             					
	CycleTime												: LREAL := 0.0;		// controller cycle time in seconds [s]					
	Kp														: LREAL := 0.0;		// proportional gain Kp	(P)								
	Tn														: LREAL := 0.0;		// integral gain Tn (I) [s]								
	Tv														: LREAL := 0.0;		// derivative gain Tv (D-T1) [s]						
	Td														: LREAL := 0.0;		// derivative damping time Td (D-T1) [s]				
	InnerWindow												: LREAL := 0.0;		// inner window for reduced I-part (dE-window)			
	OuterWindow												: LREAL := 0.0;		// outer window for disabling I-part (dE-window)		
END_VAR
VAR_OUTPUT
	Q														: LREAL := 0;		// controller output command							
	Deviation												: LREAL := 0.0;		// Setpoint deviation									
	MinLimit												: BOOL := FALSE;	// minimum limiting active ? [TRUE/FALSE] -> ARW		
	MaxLimit												: BOOL := FALSE;	// maximum limiting active ? [TRUE/FALSE] -> ARW		
	ARWActive												: BOOL := FALSE;	// ARW actice ? [TRUE/FALSE] -> freeze I-part			
	Error													: BOOL := FALSE;	// Rising edge of Error informs that an error occurred during the execution of the Function Block 							
	ErrorId													: UDINT := 0;		// Error identification 		
END_VAR                         							
VAR_OUTPUT CONSTANT                   							
	ERR_NOERROR												: UDINT := 0;		// no error												
	ERR_NOINIT												: UDINT := 1;		// no initialization done								
	ERR_INVALIDPARAM										: UDINT := 2;		// invalid parameter								
	ERR_INVALIDCYCLETIME									: UDINT := 3;		// invalid cycle time									
END_VAR
VAR
	// STATIC VARIABLE
	// Internal Variable
	fE														: LREAL := 0.0;		// error input											
	fE_1													: LREAL := 0.0;		// error input z^(-1)									
	fY														: LREAL := 0.0;		// control output										
	fY_1													: LREAL := 0.0;		// control output  z^(-1)								
	fYP														: LREAL := 0.0;		// P-part												
	fYI														: LREAL := 0.0;		// I-part												
	fYI_1													: LREAL := 0.0;		// I-part  z^(-1)										
	fYD														: LREAL := 0.0;		// D-T1-part										
	fYD_1													: LREAL := 0.0;		// D-T1-part  z^(-1)									
	// Internal Parameter
	bIsInitDone												: BOOL	:= FALSE;	// is controller init done ?							
	bInitMem												: BOOL	:= FALSE;	// reset flag											
	bIsIPart												: BOOL	:= FALSE;	// I-part active ?										
	bIsDPart												: BOOL	:= FALSE;	// D-part active ?										
	bIsDAutoScaling											: BOOL	:= FALSE;	// autoscaling for D-part done ?						
	bIsOuterWnd												: BOOL	:= FALSE;	// I-part active and outer window unequal zero ?		
                                							
	fDi														: LREAL	:= 0.0;		// internal I param										
	fDd														: LREAL	:= 0.0;		// internal D param										
	fCd														: LREAL	:= 0.0;		// internal D param										
	fCycleTime												: LREAL	:= 0.0;		// controller cycle time [s]
	MemSyncValue											: LREAL	:= 0.0;
	rtSync													: r_trig;
	rtReset													: r_trig;
END_VAR

(* controller init *)
rtReset(CLK := ResetTrig);
IF rtReset.Q OR NOT bIsInitDone OR NOT Enable 
THEN
	reset();
	RETURN;
END_IF

(* 1. check for initialisation flag *)
IF bIsInitDone 
THEN
	ErrorID 												:= ERR_NOERROR;
ELSE                                    					
	Error 													:= TRUE;
	ErrorID 												:= ERR_NOINIT;
END_IF

(* 2. controller synchronization flag => look at the end of FB *)
(* I-part *)
IF( Tn > 0.0 ) 
THEN
	fDi 												:= (Kp * fCycleTime) / (2.0 * Tn);
	bIsIPart											:= TRUE;
ELSE                                    				
	fDi 												:= 0.0;
	bIsIPart 											:= FALSE;
END_IF

(* D-part *)
IF	( Tv > 0.0 ) AND (Td > 0.0) 
THEN
	(* autoscaling necessary if (Td < CycleTime) or (Tv < Td)	*)
	(* if (Td < CycleTime) => (Td = CycleTime)					*)
	IF	( Td < fCycleTime ) 
	THEN(* autoscaling for D-part *)
		bIsDAutoScaling									:= TRUE;
		fDd 											:= (Kp * Tv) / (fCycleTime + fCycleTime / 2.0);
		fCd 											:= (fCycleTime / 2.0) / (fCycleTime + fCycleTime / 2.0);
	ELSE(* normal calculation, no autoscaling for D-part *)
		bIsDAutoScaling									:= FALSE;
		fDd 											:= (Kp * Tv) / (Td + fCycleTime / 2.0);
		fCd 											:= (Td - fCycleTime / 2.0) / (Td + fCycleTime / 2.0);
	END_IF;                             				
	bIsDPart 											:= TRUE;                   				
ELSE                                    				
	fDd													:= 0.0;
	fCd 												:= 0.0;
	bIsDPart 											:= FALSE;
END_IF;                                 				
                                        				
                                        				
(* 3. save old variable *)              				
fE_1													:= fE;
fY_1													:= fY;
fYI_1													:= fYI;
fYD_1													:= fYD;
                                        				
(* 4. set error/deviation input *)      				
Deviation												:= SetValue - ActValue;
fE														:= Deviation;  
                                     				
(* 5. YP-part *)                        	
fYp														:= Kp * fE;
                                        				
(* 6. YI-part *)                        				
IF bIsIPart                             				
THEN                                    				
	IF	( MinLimit                      				
		AND (fE < 0.0) )                				
	THEN                                				
		ARWActive										:= TRUE;
		fYI												:= fYI_1;						(* freeze I-part *)
	ELSIF	( MaxLimit                  				
			AND (fE > 0.0) )            				
	THEN                                				
		ARWActive										:= TRUE;
		fYI												:= fYI_1;						(* freeze I-part *)
	ELSE
		ARWActive										:= FALSE;
		(* fYI		:= fYI_1 + fDi * (fE + fE_1); *)					(* normal I-part calculation *)

		(* reduce I-part in the inner window *)
		IF ( ABS( fE ) < InnerWindow ) 
		THEN
			fYI 						:= fYI_1 + fDi * (fE + fE_1) * (ABS( fE ) / InnerWindow);(* reduced I-part *)
		ELSIF ( bIsOuterWnd AND ( ABS( fE ) > OuterWindow ) ) 
		THEN
			fYI											:= fYI_1;						(* freeze I-part in outer window *)
		ELSE                            				
			fYI 										:= fYI_1 + fDi * (fE + fE_1);	(* normal I-part calculation *)
		END_IF                          				
                                        				
	END_IF                              				
ELSE                                    				
	ARWActive											:= FALSE;
	fYI													:= 0.0;
END_IF                                  				
                                        	
(* 7. YD-part *)                        	
IF bIsDPart THEN                        	
	fYD													:=  fCd * fYD_1 + fDd * (fE - fE_1);
ELSE                                    				
	fYD													:= 0.0;
END_IF                                  				
                                        				
(* 8. Ysum = YP + YI + YD *)            				
fY														:= fYP + fYI + fYD;

(* 2. synchronization: Bumpless Init Without Abrupt Change Of Y(t) *)
rtSync(CLK := Sync);
IF 	ManualOn 
	OR rtSync.Q 
THEN
	Synchronize(SEL(ManualOn,SyncValue,ManualValue));
END_IF                                  				
                                        				
(* 9. check for output limiting *)      				
IF ( fY >= MaxOutput )                  				
THEN                                    				
	fY													:= MaxOutput;
	MinLimit											:= FALSE;
	MaxLimit											:= TRUE;
ELSIF ( fY <= MinOutput )               				
THEN                                    	
	fY													:= MinOutput;
	MinLimit											:= TRUE;
	MaxLimit											:= FALSE;
ELSE                                    				
	MinLimit											:= FALSE;
	MaxLimit											:= FALSE;
END_IF

(* 10. set controller output *)
Q 														:= fY;

(**********************************************************************************)

METHOD PUBLIC reset : BOOL; //Return value = TRUE if execution finished
VAR_INPUT
END_VAR
(* reset internal and external variables *)

fE															:= fE_1		:= 0.0;
fY															:= fY_1		:= 0.0;
fYP															:= 0.0;
fYI															:= fYI_1	:= 0.0;
fYD															:= fYD_1	:= 0.0;
bIsInitDone													:= FALSE;
bIsIPart													:= FALSE;
bIsDPart													:= FALSE;
ARWActive													:= FALSE;
bIsDAutoScaling												:= FALSE;
bIsOuterWnd													:= FALSE;
Q															:= 0.0;
MinLimit													:= FALSE;
MaxLimit													:= FALSE;
Error 														:= FALSE;
                            								
(* ??? set fE=fCtrlInput und fE_1=fCtrlInput ??? *)
(*	fE	:=  fCtrlInput; *)

(* read PLC cycle time for discreete calculation *)
(*	fCycleTime	:=	DINT_TO_REAL( GetScanTime( dummyInVar:= TRUE ) ) * 0.000001; *)
fCycleTime													:= CycleTime;

(* check cycle time parameter: (CycleTime > 0 AND CycleTme <= 60) *)
IF (fCycleTime <= 0) OR (fCycleTime > 60.0) 
THEN
	ErrorID 												:= ERR_INVALIDCYCLETIME;
	Error													:= TRUE;
	RETURN;
END_IF;

(* check controller parameters: (Tn, Tv, Td >= 0) *)
IF 	( (Tn < 0) 
	OR (Tv < 0) OR (Td < 0) ) 
THEN
	ErrorID 												:= ERR_INVALIDPARAM;
	Error													:= TRUE;
	RETURN;
END_IF;

(* check controller parameters: (MinOutput > MaxOutput) *)
IF ( MinOutput > MaxOutput ) 
THEN
	ErrorID 												:= ERR_INVALIDPARAM;
	Error													:= TRUE;
	RETURN;
END_IF;

(* check inner and outer window parameters: outer window must be greater than the inner window *)
IF((bIsIPart) AND ( OuterWindow > 0.0 )) 
THEN
	IF (InnerWindow > OuterWindow) 
	THEN
		ErrorId 											:= ERR_INVALIDPARAM;
		Error												:= TRUE;
		RETURN;
	END_IF;
	bIsOuterWnd 											:= TRUE;
END_IF;

(* set internal init flag *)
bIsInitDone													:= TRUE;
Q		 													:= MinOutput;
reset													:= TRUE;
END_METHOD

METHOD PUBLIC synchronize : BOOL  //Return value = TRUE if execution finished
VAR_INPUT 
	IN											:	LREAL;
END_VAR
	MemSyncValue										:= IN;
	
	(* Demand:  SyncValue != Ysum  with  SyncValue = Ysum = YP + YI + YD  =>  YI = SyncValue - Yp - Yd *)
	IF 	( bIsIPart = TRUE ) 
	THEN	(* I-part exists independent from the D-part *)
		(* Normal:  fYI = fYI_1 + fDi * (fE + fE_1) *)
		fYD 											:= fYD_1	:= 0.0;								
		fYI												:= fYI_1	:= MemSyncValue - fYP - fYD;	
		fY												:= MemSyncValue;
	ELSIF ( bIsDPart = TRUE ) 
	THEN	(* no I-part available, only D-part exits *)
		(* Normal:  fYD = fCd * fYD_1 + fDd * (fE - fE_1) *)
		(* fYD := fYD_1 := (fSyncValue - fYP - fYI) / fCd;*)(* 1) pre-calculation for the next cycle; fYI must be zero because there exists no I-part *)
		fYD												:= fYD_1	:= (MemSyncValue - fYP - fYI);		(* 2) fYI must be zero because there exists no I-part *)
		fY												:= MemSyncValue;
	END_IF                              				
	
	Synchronize											:= TRUE;
END_METHOD

END_FUNCTION_BLOCK

// POUs/ControllerTools/PT1Filter
//Low pass filter with a programmable time Tn and factor Kp.
FUNCTION_BLOCK PT1Filter
VAR_INPUT
	Enable													:	BOOL ; 	// FB will be processed as long as enable is TRUE 
	In														:	LREAL := 0.0;	// Actual value
	ResetTrig												:	BOOL ; 	// The function block will be reset with a rising edge 
	Sync													:	BOOL ; 	// Synchronise In to Q - equivalent to Synchronize method
	Kp														:	LREAL := 1.0; 	// Gain
	Tn														:	TIME := T#1S; 	// Integral time 
	Cycletime 												:	TIME := T#10MS;	// cycletime 
END_VAR	            										
VAR_OUTPUT          										
	Q														: LREAL;			// Output
	Error													: BOOL;				// Rising edge of Error informs that an error occurred during the execution of the Function Block 
END_VAR             										
VAR                 	
	Q_old													: LREAL;
END_VAR

(**************************************************************************************
	formula: 
	y(k) = [1-T/T1]	* y(k-1)
			+ T/T1		* v 		* e(k) 
*************************************************************************************)

	Error 													:= Cycletime = T#0MS OR  tn = T#0MS OR Kp = 0.0;
                            								
	IF Enable               								
		AND NOT Error       								
	THEN                    								
		Q 													:=  (1- TIME_TO_LREAL(Cycletime) / TIME_TO_LREAL(Tn))	* Q_old
															 	+ TIME_TO_LREAL(Cycletime) / TIME_TO_LREAL(Tn)	* Kp		* In;
		Q_Old 												:= Q;
	ELSE //Hold
		;
	END_IF

	IF ResetTrig
	THEN
		reset();
	ELSIF Sync
	THEN
		Synchronize(IN);
	END_IF

(************************************************************************************)

METHOD reset : BOOL //Return value = TRUE if execution finished
VAR_INPUT
END_VAR
Q := Q_old 				:= 0.0;
reset				:= TRUE;
END_METHOD

METHOD PUBLIC synchronize : BOOL //Return value = TRUE if execution finished
VAR_INPUT
	IN						:	LREAL;
END_VAR
Q 	:= Q_Old 	 := IN;
Synchronize		:= TRUE;
END_METHOD

END_FUNCTION_BLOCK

// POUs/ControllerTools/signum
//LREAL Signum function
FUNCTION signum : LREAL
VAR_INPUT
	IN		:	LREAL;
END_VAR
VAR
END_VAR

IF IN = 0.0
THEN
	SIGNUM		:= 0.0;
ELSIF IN > 0.0
THEN
	SIGNUM		:= 1.0;
ELSE
	SIGNUM	 	:= -1.0;
END_IF

END_FUNCTION

// POUs/ControllerTools/SlewRateLimitter
//LREAL Slew rate limitter with a timebased change rate
FUNCTION_BLOCK SlewRateLimitter
VAR_INPUT
	IN														: LREAL := 0.0;	 //Actual value
	Sync													: BOOL := FALSE; //Sync signal sets IN to Q	
	Cycletime												: LREAL := 0.001; //cycletime in ms
	Rate													: LREAL := 1.0;	 // changes per second
END_VAR                 									
VAR_OUTPUT              									
	Q														: LREAL := 0.0;   //Output
END_VAR                 									
VAR                     	
	x														: LREAL := 0.0;
END_VAR

//Based on MC_AxUtiSlewRateLimitter_BkPlcMc from TcPlcLibHydraulics , Author WOs
IF Cycletime <= 0.0001 OR Rate <= 0.0 OR Sync
THEN
	Q														:= IN;
ELSE                    									
	x														:= Cycletime * Rate;
	IF ABS(IN) > X OR ABS(Q > In)
	THEN //Start ramping only after In is greater than Rate and as long as Q is greater (if In jumps to zero)
		Q													:= Q + LIMIT(-x , IN - Q , x); 		
	ELSE
		Q													:= In;
	END_IF
END_IF

METHOD PUBLIC synchronize : BOOL //Return value = TRUE if execution finished
VAR_INPUT
	IN														:	LREAL;
END_VAR
Q 															:= IN;
Synchronize 												:= TRUE;
END_METHOD

END_FUNCTION_BLOCK

// POUs/ControllerTools/SlidingAverage
FUNCTION_BLOCK SlidingAverage 
VAR_OUTPUT CONSTANT 
	MIN_BUFFER												:	INT := 1;
	MAX_BUFFER												:	INT := PARAM.SLIDING_AVERAGE_MAX_ENTRYS;
END_VAR
VAR_INPUT
	In														: LREAL := 0.0;			//Actual value 
	ResetTrig												: BOOL := FALSE;		//Reset average buffer
	MaxNoOfValues											: DINT := PARAM.SLIDING_AVERAGE_MAX_ENTRYS;//Buffer limit if value is smaller than MAX_BUFFER
	SampleTime												: TIME := T#0MS;
END_VAR                 									
VAR_OUTPUT              									
	Q														: LREAL := 0.0;			//Average value
	Derivative												: LREAL := 0.0;			//
	ActIdx													: DINT := 1; 			//rotating count of buffer 
	Buffer													: ARRAY [MIN_BUFFER..MAX_BUFFER] OF LREAL;
END_VAR                 									
VAR           
	MinIdx													: DINT := MIN_BUFFER;   
	MaxIdx													: DINT := 0;       									
	Count													: DINT := 0; // limited count 
	pBuffer													: POINTER TO LREAL := 0;
	pIdx													: POINTER TO LREAL := 0;
	IdxOld													: DINT := 1;
	ftotal													: LREAL;
	fttotal													: LREAL;
	tonSampleTimer											: ton;
END_VAR


IF ResetTrig THEN reset(); RETURN; END_IF

pBuffer														:= ADR(Buffer);
MaxIdx														:= LIMIT(MIN_BUFFER, TO_INT(MaxNoOfValues), MAX_BUFFER);

IF(ActIdx>MaxIdx)
THEN
	ActIdx													:= MinIdx;
END_IF                      								
IF(ActIdx<MinIdx)           								
THEN                        								
	ActIdx													:= MaxIdx;
END_IF                      								
                            								
IF(ActIdx>MaxIdx)           								
THEN                        								
	Q														:= IN; (* Puffer-Indices sind unsinnig *)
ELSIF(pBuffer=0)            								
THEN                        								
	Q														:= IN; (* Puffer-Adresse ist unsinnig *)
ELSE            
	tonSampleTimer(IN := SampleTime > T#0MS, PT :=  SampleTime);
	IF NOT tonSampleTimer.IN OR tonSampleTimer.Q    
	THEN   			
		tonSampleTimer(IN := FALSE);	
		
		Count												:= MIN(Count, MaxIdx - MinIdx + 1);
		IdxOld												:= ActIdx - Count;
															
		IF(IdxOld<MinIdx)      								
		THEN                    							
			IdxOld											:= IdxOld + MaxIdx - MinIdx + 1;
		END_IF                  	                        
									                        
		IF(ActIdx=MinIdx)       	                        
		THEN                    	                        
			fttotal											:= 0.0;
		END_IF                  							
															
		IF(Count<1)            								
		THEN                    							
			ftotal := Derivative 							:= 0.0;	(* first cycle *)
		END_IF                  							
															
		pIdx												:= pBuffer + ((ActIdx - MinIdx) * SIZEOF(LREAL));
									                        
		IF(Count = (MaxIdx - MinIdx + 1))                   
		THEN                                                
			Derivative										:= (IN - pIdx^) / DINT_TO_LREAL(Count);
			ftotal											:= ftotal-pIdx^;		(* buffer is filled at least once *)
		END_IF                  							
		pIdx^												:=IN;
		fttotal												:=fttotal + IN;
		ftotal												:=ftotal + IN;
															
		ActIdx												:=ActIdx + 1;
									                        
		IF(ActIdx > MaxIdx)                                 
		THEN                                                
			(* swapping *)                                  
			ftotal											:= fttotal;
			ActIdx											:= MinIdx;
		END_IF                                              
		                                                    
		Count												:= MIN(Count + 1, MaxIdx - MinIdx + 1);
															
		Q													:=ftotal / DINT_TO_LREAL(Count);
	END_IF
END_IF

METHOD PUBLIC reset : BOOL //Return value = TRUE if execution finished
VAR_INPUT
END_VAR
Q															:=0.0;
Derivative													:=0.0;
ActIdx														:=MIN_BUFFER;	(* rotating count *)
Count														:=0;			(* limited count *)
                        									
                        									
IdxOld														:=1;
                        	
ftotal														:=0.0;
fttotal														:=0.0;
MEMSET(ADR(Buffer), 0 , SIZEOF(Buffer));
reset													:= TRUE;
END_METHOD

END_FUNCTION_BLOCK

// POUs/ControllerTools/SlidingAverageExt
//LREAL Sliding average with dynamic allocation of memory according MaxNoofValues 
{attribute 'enable_dynamic_creation'}
FUNCTION_BLOCK SlidingAverageExt 
VAR_INPUT
	In														: LREAL := 0.0;			//Actual value 
	ResetTrig												: BOOL ;		//Reset average buffer
	MaxNoOfValues											: DINT (0..10000) := 0;//Size of buffer (Array size) needs to get assigend in declaration
	SampleTime												: TIME := T#0MS;
END_VAR                 									
VAR_OUTPUT              									
	Q														: LREAL := 0.0;			//Average value
	Derivative												: LREAL := 0.0;			//
	ActIdx													: DINT := 1; 			//rotating count of buffer 
END_VAR                 									
VAR       
	MaxIdx													: DINT := 0;      
	MinIdx													: DINT := 1;        									
	Count													: DINT := 0; // limited count 
	pBuffer													: POINTER TO LREAL := 0;
	pIdx													: POINTER TO LREAL := 0;
	IdxOld													: DINT := 1;
	ftotal													: LREAL;
	fttotal													: LREAL;
	tonSampleTimer											: ton;
END_VAR

(* be sure to have nIdx inside MinIdx..MaxIdx *)
IF pBuffer = 0 AND MaxNoOfValues > 0
THEN //Alocate buffer memory
	pBuffer 												:= __NEW(LREAL,TO_UDINT(MaxNoOfValues)); 	
	IF NOT PARAM.ENABLE_DEBUG_MSG_DYNAMIC_MEM_ALLOCATION
	THEN 
		;
	ELSIF MaxIdx = 0 
	THEN
		AdsLogHint('EngineeringToolbox | FB SlidingAverageExt | An instance allocated %s bytes from the dynamic memory of the ADS router memory pool', TO_STRING(MaxNoOfValues * SIZEOF(LREAL)));	
	ELSE //Allocation of additional memory space
		AdsLogWarn('EngineeringToolbox | FB SlidingAverageExt | Value of "MaxNoOfValues" changed and one instance allocated additional %s bytes from the dynamic memory of the ADS router memory pool', TO_STRING(MaxNoOfValues * SIZEOF(LREAL)));
	END_IF
	MinIdx													:= 1;
	MaxIdx													:= MaxNoOfValues;
ELSIF MaxNoOfValues <> MaxIdx OR MaxNoOfValues = 0
THEN
	reset();
	FB_exit(FALSE);
	RETURN;
END_IF

IF ResetTrig THEN reset(); RETURN; END_IF

IF(ActIdx>MaxIdx)
THEN
	ActIdx													:= MinIdx;
END_IF                      								
IF(ActIdx<MinIdx)           								
THEN                        								
	ActIdx													:= MaxIdx;
END_IF                      								
                            								
IF(ActIdx>MaxIdx)           								
THEN                        								
	Q														:= IN; (* Puffer-Indices sind unsinnig *)
ELSIF(pBuffer=0)            								
THEN                        								
	Q														:= IN; (* Puffer-Adresse ist unsinnig *)
ELSE       
	tonSampleTimer(IN := SampleTime > T#0MS, PT :=  SampleTime);
	IF NOT tonSampleTimer.IN OR tonSampleTimer.Q    
	THEN   			                                        
		tonSampleTimer(IN := FALSE);	                 							
		Count												:= MIN(Count, MaxIdx - MinIdx + 1);
		IdxOld												:= ActIdx - Count;
															
		IF(IdxOld<MinIdx)      								
		THEN                    							
			IdxOld											:= IdxOld + MaxIdx - MinIdx + 1;
		END_IF                  	                        
									                        
		IF(ActIdx=MinIdx)       	                        
		THEN                    	                        
			fttotal											:= 0.0;
		END_IF                  							
															
		IF(Count<1)            								
		THEN                    							
			ftotal := Derivative 							:= 0.0;	(* first cycle *)
		END_IF                  							
															
		pIdx												:= pBuffer + ((ActIdx - MinIdx) * SIZEOF(LREAL));
									                        
		IF(Count = (MaxIdx - MinIdx + 1))                   
		THEN                                                
			Derivative										:= (IN - pIdx^) / DINT_TO_LREAL(Count);
			ftotal											:= ftotal-pIdx^;		(* buffer is filled at least once *)
		END_IF                  							
		pIdx^												:=IN;
		fttotal												:=fttotal + IN;
		ftotal												:=ftotal + IN;
															
		ActIdx												:=ActIdx + 1;
									                        
		IF(ActIdx > MaxIdx)                                 
		THEN                                                
			(* swapping *)                                  
			ftotal											:= fttotal;
			ActIdx											:= MinIdx;
		END_IF                                              
		                                                    
		Count												:= MIN(Count + 1, MaxIdx - MinIdx + 1);
															
		Q													:=ftotal / DINT_TO_LREAL(Count);
	End_If
END_IF

METHOD FB_exit : BOOL 
VAR_INPUT
	bInCopyCode : BOOL; // if TRUE, the exit method is called for exiting an instance that is copied afterwards (online change).
END_VAR
IF NOT bInCopyCode AND pBuffer <> 0
THEN //Release memory in case the PLC stopps
	__DELETE(pBuffer);
	MaxIdx								:= 0;
END_IF
END_METHOD

METHOD PUBLIC reset : BOOL //Return value = TRUE if execution finished
VAR_INPUT
END_VAR
Q															:=0.0;
Derivative													:=0.0;
ActIdx														:=1;			(* rotating count *)
Count														:=0;			(* limited count *)
                        									
                        									
IdxOld														:=1;
                        	
ftotal														:=0.0;
fttotal														:=0.0;


IF pBuffer <> 0
THEN
	MEMSET(pBuffer, 0 , SIZEOF(pBuffer^));
END_IF	

reset														:= TRUE;
END_METHOD

END_FUNCTION_BLOCK

// POUs/Logging/adsLogHint
{attribute 'no_check' := ''}
//Writes a string as a hint message into the TwinCAT AMS Logger and Windows Event Log with an possible argument
//Please see Beckhoff information system "ADSLOGxxxx" for detailed information.
//Intention of this function is to use the handy ADSLOGxxxx with a predefined msgCtrlMask of "ADSLOG_MSGTYPE_STRING OR ADSLOG_MSGTYPE_HINT OR ADSLOG_MSGTYPE_LOG"
FUNCTION adsLogHint : DINT//Write hint message into ADS log windows - Return value will be error code or 0 if OK
VAR_INPUT               											
	MsgFmtStr												:	T_MaxString; ///Message text with %s as placeholder for StrArg
(*	dintArg													:	DINT; //DINT argument for message - to be replaced by %d *) 
	StrArg													:	T_MaxString; //String argument for message - to be replaced by %s
(*	realArg													:	LREAL; //LREAL argument for message - to be replaced by %f *) 
END_VAR
VAR
	msgCtrlMask												:	DWORD; (* 	ADSLOG_MSGTYPE_HINT Meldungstyp ist Hinweis.
																				ADSLOG_MSGTYPE_WARN Meldungstyp ist Warnung.  
																				ADSLOG_MSGTYPE_ERROR Meldungstyp ist Fehler.  
																				ADSLOG_MSGTYPE_LOG Meldung wird in das Logbuch geschrieben.  
																				ADSLOG_MSGTYPE_MSGBOX Meldung wird in einer Messagebox ausgegeben.  
																				ADSLOG_MSGTYPE_RESOURCE Meldung wird aus einer Ressource-Datei geholt. (wird momentan nicht  unterstützt)  
																				ADSLOG_MSGTYPE_STRING 	Meldung ist direkt angegebener String (default).  *)	
END_VAR

(* create fixed message ctrl mask **********************************)
	msgCtrlMask												:= ADSLOG_MSGTYPE_STRING OR ADSLOG_MSGTYPE_HINT OR ADSLOG_MSGTYPE_LOG;

(* write string which includes a floating-number ******************)
(*	AdsLogHint 												:= ADSLOGLREAL(msgCtrlMask, msgFmtStr, realArg); *)
	
(* write string which includes a DINT-number *******************)
(*	AdsLogHint 												:= ADSLOGDINT(msgCtrlMask, msgFmtStr, dintArg); *)

(* write string which includes an other string e.g. 'hallo: %s what's up' ***************)
	adsLogHint 												:= ADSLOGSTR(msgCtrlMask, msgFmtStr,strArg); 

(*****************************************************)

END_FUNCTION

// POUs/Logging/adsLogWarn
{attribute 'no_check' := ''}
//Writes a string as a warining message into the TwinCAT AMS Logger and Windows Event Log with an possible argument
//Please see Beckhoff information system "ADSLOGxxxx" for detailed information.
//Intention of this function is to use the handy ADSLOGxxxx with a predefined msgCtrlMask of "ADSLOG_MSGTYPE_STRING OR ADSLOG_MSGTYPE_WARN OR ADSLOG_MSGTYPE_LOG"
FUNCTION adsLogWarn : DINT//Write warning message into ADS log windows - Return value will be error code or 0 if OK
VAR_INPUT               											
	MsgFmtStr												:	T_MaxString; //Message text with %s as placeholder for StrArg
(*	dintArg													:	DINT; //DINT argument for message - to be replaced by %d *) 
	StrArg													:	T_MaxString; //String argument for message - to be replaced by %s
(*	realArg													:	LREAL; //LREAL argument for message - to be replaced by %f *) 
END_VAR
VAR
	msgCtrlMask												:	DWORD; (* 	ADSLOG_MSGTYPE_HINT Meldungstyp ist Hinweis.
																				ADSLOG_MSGTYPE_WARN Meldungstyp ist Warnung.  
																				ADSLOG_MSGTYPE_ERROR Meldungstyp ist Fehler.  
																				ADSLOG_MSGTYPE_LOG Meldung wird in das Logbuch geschrieben.  
																				ADSLOG_MSGTYPE_MSGBOX Meldung wird in einer Messagebox ausgegeben.  
																				ADSLOG_MSGTYPE_RESOURCE Meldung wird aus einer Ressource-Datei geholt. (wird momentan nicht  unterstützt)  
																				ADSLOG_MSGTYPE_STRING 	Meldung ist direkt angegebener String (default).  *)	
END_VAR

(* create fixed message ctrl mask **********************************)
	msgCtrlMask												:= ADSLOG_MSGTYPE_STRING OR ADSLOG_MSGTYPE_WARN OR ADSLOG_MSGTYPE_LOG;

(* write string which includes a floating-number ******************)
(*	AdsLogWarn 												:= ADSLOGLREAL(msgCtrlMask, msgFmtStr, realArg); *)
	
(* write string which includes a DINT-number *******************)
(*	AdsLogWarn 												:= ADSLOGDINT(msgCtrlMask, msgFmtStr, dintArg); *)

(* write string which includes an other string e.g. 'hallo: %s what's up' ***************)
	adsLogWarn 												:= ADSLOGSTR(msgCtrlMask, msgFmtStr,strArg); 

(*****************************************************)

END_FUNCTION

// POUs/ControllerTools/ThreePointController
//Three point controller with lreal output
//The On-Values must be greater then the Off-Values. The difference is equivalent to the hysteresis-value
FUNCTION_BLOCK ThreePointController 
VAR_INPUT
	Enable													: BOOL := TRUE;		//Enable controller	
	SetValue												: LREAL := 0.0;		//Setpoint value
	ActValue												: LREAL := 0.0;		//Actual value
	
	Sync													: BOOL := FALSE; 	//Synchronization flag for bumpless initialisation		
	SyncValue												: LREAL := 0.0; 	//Syncronization value for bumpless init.			
	MinOutput												: LREAL := 0.0; 	//Controller minimum analog output			
	MaxOutput												: LREAL := 100.0;	//Controller maximum analog output (Limitation is switched off at 0.0) 			

	FeedPlus												: BOOL := TRUE;		//Release for controller plus 
	FeedMinus												: BOOL := TRUE;		//Release for controller minus 
	                                						
	ManualOn												: BOOL := FALSE;	//Manual mode on - set analog output to ManualValue
	ManualValue												: LREAL	:= 0.0;		//Analog output in manual mode
	ManualPlus												: BOOL := FALSE;	//Manual control of digital plus output	
	ManualMinus												: BOOL := FALSE;	//Manual control of digital minus output	
                                    						
	Stepwide												: LREAL := 1.0; 	//Stepwidth analog output
	Breaktime												: TIME := T#500MS; 	//Breaktime after a change of output
	DriveTime												: TIME := T#500MS; 	//Drivetime for digital outputs  
	                                					
	PlusOn													: LREAL := 5.0;		//Derivate hysteresis to increase the controller output (need to be greater than PlusOff , Plus or Minus pair need to be less the zero)  
	PlusOff													: LREAL := 3.0;		//Derivate hysteresis to switch off the controller output (need to be smaller than PlusOn , Plus or Minus pair need to be less the zero  
	MinusOff												: LREAL := -3.0;	//Derivate hysteresis to switch the controller output (need to be greater smaller than MinusOn , Plus or Minus pair need to be less the zero) 
	MinusOn													: LREAL := -5.0;	//Derivate hysteresis to decrease the controller output (need to be greater than MinusOff , Plus or Minus pair need to be less the zero)
END_VAR                             						
VAR_OUTPUT	   
	Q														: LREAL; 			//Analog controller output
	Q_Plus													: BOOL;				//Digital controller output
	Q_Minus													: BOOL;				//Digital controller output
	Deviation												: LREAL;			//deviation between actual value and setpoint (Deviation = SetValue - ActValue)
	DeadZone												: LREAL;			//Active dead zone based on PlusOn/Off and MinusOn/Off values
	BreakTimeRunning										: BOOL;				//Controller is on hold - Break time running 
	DriveTimeRunning										: BOOL;				//Controller is active 
	Error													: BOOL;             //Error occured       						
END_VAR                             						
VAR 
//local variables *********************************************************          
	state													: INT;     
	MemPlus													: BOOL;
	MemMinus												: BOOL;
	Cooling													: BOOL;      

//Trigger ****************************************************************           						
	rtSync													: r_trig;	
	
//timer ******************************************************************
	tonBreakTime											:	ton;
	tonDriveTime											:	ton;

	
END_VAR

(* 3 point bang-bang controller 	 							*)
(****************************************************************)

IF ABS(MinusOn) <= ABS(MinusOff) //On offset must be greater then off
	OR ABS(PlusOn) <= ABS(PlusOff) //Off offsetr must be smallet then on
	OR NOT(MinusOn > 0.0 XOR PlusOn > 0.0)//Only one offset needs to be greater then 0.0
	OR NOT(PlusOff > 0.0 XOR MinusOff > 0.0)//Only one offset needs to be greater then 0.0
	OR MinOutput > MaxOutput AND MaxOutput <> 0.0
THEN
	reset();
	Error													:= Enable;
ELSE                                            			
	rtSync(CLK := Sync);                        			
	IF rtSync.Q                                 			
	THEN                                        			
		Synchronize(SyncValue); 
	END_IF                                      			
	                                            			
	Error													:= FALSE;
	DeadZone												:= ABS(PlusOff) + ABS(MinusOff);
	Deviation												:= SetValue - ActValue; 
	Cooling													:= PlusOn < 0.0 AND MinusOn > 0.0;
		  
	//Control sequecne                                      			
	CASE state OF                               			
	0:                                          			
		//Check wheter controller needs to start 
		IF ManualON                             			
		THEN                                    			
			MemMinus := MemPlus								:= FALSE;
			Q												:= ManualValue;
		ELSIF NOT Enable                        			
		THEN                                    			
			reset();
		ELSIF(Q < MaxOutput OR MaxOutput = 0.0)       
			AND FeedPlus    			
			AND(                                			
			Deviation > PlusOn AND NOT Cooling     			
			OR  Deviation < PlusOn AND Cooling)     			
		THEN // greatest Plusitive deviatoin      			
			MemPlus											:= TRUE;
			MemMinus										:= FALSE;
		ELSIF(Q > MinOutput OR MaxOutput = 0.0)    
			AND FeedMinus      			
			AND(                                			
			Deviation < MinusOn AND NOT Cooling      	
			OR Deviation > MinusOn AND Cooling)      			
		THEN // greatest Minusative deviation     			
			MemMinus										:= TRUE;
			MemPlus											:= FALSE;
			
		ELSE
			MemPlus											:= MemPlus AND ABS(Deviation) >= ABS(PlusOff) ;
			MemMinus										:= MemMinus AND ABS(Deviation) >= ABS(MinusOff);
		END_IF              			
		                       
		//Continue to run controller up or down as long as memory is still active                  			
		IF MemMinus	                            			
		THEN                                    			
			Q												:= MAX(Q - Stepwide, MinOutput);
			state											:= 1;
		ELSIF MemPlus                            			
		THEN                                    			
			Q												:= MIN(Q + Stepwide, MaxOutput);
			state											:= 1;
		ELSE                                    			
			Q												:= LIMIT(MinOutput, Q, MaxOutput);
		END_IF		
			
	1: //start drive time 
		tonDriveTime(IN := FALSE); tonBreakTime(IN := FALSE);
		IF DriveTime > T#0MS
		THEN
			tonDriveTime(IN := TRUE, PT := DriveTime);
			state											:= 2;
		ELSIF BreakTime > T#0MS
		THEN
			tonBreakTime(IN := TRUE, PT := BreakTime);	
			state											:= 3;	
		ELSE
			state											:= 0;			
		END_IF
				                    			
	2:  //run drive time                                       			
		tonDriveTime();
		IF ManualOn
		THEN
           state											:= 0;    			
		ELSIF tonDriveTime.Q                			
		THEN
			IF BreakTime > T#0MS
			THEN
				tonBreakTime(IN := TRUE, PT := BreakTime);
				state										:= 3;
			ELSE
				state										:= 0;				
			END_IF				             	
		END_IF     
                    
	3: //run break time 
		tonBreakTime();
		IF ManualOn OR tonBreakTime.Q  
		THEN
           state											:= 0;    			
		END_IF	
	END_CASE                                    			
	
	//status
	DriveTimeRunning										:= state = 2;
	BreakTimeRunning										:= state = 3;
                                            			                      			                                                		
	//setting ouputs
	Q_Minus 												:= FeedMinus AND Enable
																AND(
																MemMinus AND DriveTimeRunning 
																OR ManualOn AND ManualMinus) ;
										
	Q_Plus				 									:= FeedPlus AND Enable
																AND(
																MemPlus AND DriveTimeRunning
																OR ManualOn AND ManualPlus) ;
																						
END_IF

METHOD PUBLIC reset : booL //Return value = TRUE if execution finished
VAR_INPUT
END_VAR
Q												:= MinOutput;
MemMinus := MemPlus								:= FALSE;
state											:= 0;

Q_Plus											:= FALSE;
Q_Minus											:= FALSE;
Error											:= FALSE;
Deviation										:= 0.0;
DeadZone										:= 0.0;
BreakTimeRunning								:= FALSE;
DrivetimeRunning								:= FALSE;

reset										:= TRUE;
END_METHOD

METHOD PUBLIC synchronize : BOOL //Return value = TRUE if execution finished
VAR_INPUT
	IN											:	LREAL;
END_VAR
Q								:= LIMIT(MinOutput,IN,MaxOutput);
Synchronize						:= TRUE;
END_METHOD

END_FUNCTION_BLOCK

// POUs/DataBuffer/Fifo/Fifo
//Fifo base control template with external memory based of FifoBase
FUNCTION_BLOCK Fifo EXTENDS FifoBase
VAR_INPUT
END_VAR
VAR_OUTPUT
END_VAR
VAR
END_VAR

;

//Clear out one entry from the Fifo buffer
METHOD PUBLIC clear : BOOL //TRUE if method was successful
VAR_INPUT
	EntryNo													:	UDINT;
	pMemory													: 	POINTER TO BYTE := 0;
	SizeOfMemory											: 	UDINT := 0;
END_VAR             										
VAR                 										
END_VAR
Clear := SUPER^._Clear(EntryNo,pMemory,SizeOfMemory);
END_METHOD

//Clear out defined data set from the Fifo buffer
METHOD PUBLIC clearByDataSet : BOOL //TRUE if method was successful
VAR_INPUT
	pData													: 	POINTER TO BYTE := 0;
	SizeOfData												: 	UDINT := 0;										
	pMemory													: 	POINTER TO BYTE := 0;
	SizeOfMemory											: 	UDINT := 0;
END_VAR             										
VAR         
	i														:	DINT;        										
END_VAR
ClearByDataSet := SUPER^._ClearByDataSet(pData,SizeOfEntry,pMemory,SizeOfMemory);
END_METHOD

METHOD PUBLIC dequeue : BOOL //TRUE if method was successful
VAR_INPUT
	pData													: 	POINTER TO BYTE := 0;
	SizeOfData												: 	UDINT := 0;
	pMemory													: 	POINTER TO BYTE := 0;
	SizeOfMemory											: 	UDINT := 0;
END_VAR
Dequeue := SUPER^._Dequeue(pData,SizeOfEntry,pMemory,SizeOfMemory);
END_METHOD

METHOD PUBLIC enqueue : BOOL //TRUE if method was successful
VAR_INPUT
	pData													: 	POINTER TO BYTE := 0;
	SizeOfData												: 	UDINT := 0;
	pMemory													: 	POINTER TO BYTE := 0;
	SizeOfMemory											: 	UDINT := 0;
END_VAR
Enqueue := SUPER^._Enqueue(pData,SizeOfData,pMemory,SizeOfMemory);
END_METHOD

//Check wheter a value already exist
METHOD PUBLIC isEnqueued : uDINT //data exist in Fifo if reurn value <> 0, returns index of entry in buffer 
VAR_INPUT
	pData													: 	POINTER TO BYTE := 0;
	SizeOfData												: 	UDINT := 0;
	pMemory													: 	POINTER TO BYTE := 0;
	SizeOfMemory											: 	UDINT := 0;
END_VAR	
VAR
	i 														: 	DINT;
END_VAR
IsEnqueued := SUPER^._IsEnqueued(pData,SizeOfEntry,pMemory,SizeOfMemory);
END_METHOD

//Check wheter a value will be the next output of the buffer
METHOD PUBLIC isNextEntry : BOOL //Inputs value is the next output 
VAR_INPUT
	pData													: 	POINTER TO BYTE := 0;
	SizeOfData												: 	UDINT := 0;
	pMemory													: 	POINTER TO BYTE := 0;
	SizeOfMemory											: 	UDINT := 0;
END_VAR
VAR
END_VAR
IsNextEntry := SUPER^._IsNextEntry(pData,SizeOfEntry,pMemory,SizeOfMemory);
END_METHOD

METHOD PUBLIC readEntry : BOOL //TRUE if method was successful
VAR_INPUT
	idx														:	UDINT;
	pData													: 	POINTER TO BYTE := 0;
	SizeOfData												: 	UDINT := 0;
	pMemory													: 	POINTER TO BYTE := 0;
	SizeOfMemory											: 	UDINT := 0;
END_VAR
ReadEntry := SUPER^._ReadEntry(idx,pData,SizeOfEntry,pMemory,SizeOfMemory);
END_METHOD

//Reset complete Fifo
METHOD PUBLIC reset : BOOL //TRUE if method is finnished
VAR_INPUT
	pMemory													: 	POINTER TO BYTE := 0;
	SizeOfMemory											: 	UDINT := 0;
END_VAR
reset := SUPER^._reset(pMemory,SizeOfMemory);
END_METHOD

END_FUNCTION_BLOCK

// POUs/DataBuffer/Fifo/FifoBase
//Fifo basic control template with external memory 
FUNCTION_BLOCK FifoBase
VAR_INPUT
	Overwrite												:	BOOL := FALSE; //Return value TRUE = overwrite oldest entry 
END_VAR
VAR_OUTPUT
	Count													:	UDINT := 0; //Number of entrys	
	Full													:	BOOL := FALSE; //Fifo is full
	Empty													:	BOOL := TRUE;  //Fifo is empty
END_VAR
VAR
	Interlock												:	BOOL; //Multitask interlock
	MaxEntrys												:	UDINT := 0; //Maximum number of entrys based on size of data and size of memory
	SizeOfEntry												:	UDINT := 0;
END_VAR

;

//Clear out one entry from the Fifo buffer
METHOD PROTECTED _clear : BOOL //TRUE if method was successful
VAR_INPUT
	EntryNo													:	UDINT;
	pMemory													: 	POINTER TO BYTE := 0;
	SizeOfMemory											: 	UDINT := 0;
END_VAR             										
VAR                 										
END_VAR
IF EntryNo = 0
	OR pMemory = 0
	OR SizeOfMemory = 0
THEN
	_Clear													:= FALSE;
	RETURN;
ELSIF TestAndSet(Interlock)
THEN	
	IF Empty OR EntryNo > Count
	THEN
		_Clear												:=TRUE;
	ELSE	                        						
		MaxEntrys 											:= SizeOfMemory / SizeOfEntry;	
		
		//shift datasets
		MEMMOVE(pMemory + ((EntryNo - 1) * SizeOfEntry) , pMemory + (EntryNo * SizeOfEntry)  , (Count - EntryNo) * SizeOfEntry);
		
		//delete last shifted dataset 
		MEMSET(pMemory + ((Count - 1) * SizeOfEntry),0, SizeOfEntry);

		Count 												:= MAX(0,Count - 1);
		Full 												:= FALSE;
		Empty 												:= Count = 0;
		_Clear												:= TRUE;	
	END_IF
	Interlock												:= FALSE;
ELSE
	_Clear													:= FALSE;
END_IF
END_METHOD

//Clear out defined data set from the Fifo buffer
METHOD PROTECTED _clearByDataSet : BOOL //TRUE if method was successful
VAR_INPUT
	pData													: 	POINTER TO BYTE := 0;
	SizeOfData												: 	UDINT := 0;										
	pMemory													: 	POINTER TO BYTE := 0;
	SizeOfMemory											: 	UDINT := 0;
END_VAR             										
VAR         
	i														:	UDINT;        										
END_VAR
IF 	pData = 0
	OR SizeOfData = 0
	OR pMemory = 0
	OR SizeOfMemory = 0
	OR Empty
THEN
	_ClearByDataSet											:= FALSE;
	RETURN;
ELSIF TestAndSet(Interlock)
THEN
	_ClearByDataSet											:= FALSE;
	MaxEntrys 												:= SizeOfMemory / SizeOfData;	
	FOR i := Count TO 1 BY -1
	DO
		
		IF MEMCMP(pData,pMemory + ((i - 1) * SizeOfData), SizeOfData) = 0
		THEN
			IF TO_UDINT(i) >= MaxEntrys
			THEN //Just delete the entry at the end of the list
				MEMSET(pMemory + ((i - 1) * SizeOfData),0, SizeOfData);
				Count 										:= MAX(0,Count - 1);
			ELSE //Copy the other entrys over the found one and delte the left entry from the list
				MEMMOVE(pMemory + ((i - 1) * SizeOfData),pMemory + (i * SizeOfData) , MIN(Count - i, MaxEntrys - 1) * SizeOfData);
				MEMSET(pMemory + ((Count - 1 )* SizeOfData),0, SizeOfData);
				Count 										:= MAX(0,Count - 1);
			END_IF		
			_ClearByDataSet									:= TRUE;
			Full 											:= FALSE;
			Empty 											:= Count = 0;		
			IF Empty 
			THEN
				EXIT;
			END_IF
		END_IF
	END_FOR
	Interlock												:= FALSE;
END_IF
END_METHOD

METHOD PROTECTED _dequeue : BOOL //TRUE if method was successful
VAR_INPUT
	pData													: 	POINTER TO BYTE := 0; //pointer to destination of data
	SizeOfData												: 	UDINT := 0; //Size of destination data
	pMemory													: 	POINTER TO BYTE := 0;
	SizeOfMemory											: 	UDINT := 0;
END_VAR
IF 	pData = 0
	OR SizeOfData = 0
	OR pMemory = 0
	OR SizeOfMemory = 0
	OR Empty
THEN
	_Dequeue												:= FALSE;
	RETURN;
ELSIF TestAndSet(Interlock)
THEN	
	(* copy dataset *)
	MEMMOVE(pData,pMemory + (MAX(0, (Count - 1)) * SizeOfData),SizeOfData);
	
	(* delete dataset *)
	MEMSET(pMemory + (MAX(0,(Count - 1)) * SizeOfData) ,0 ,SizeOfData);
	Count 													:= MAX(0,Count - 1);
	Full 													:= FALSE;
	Empty 													:= Count = 0;
	_Dequeue												:= TRUE;
	Interlock												:= FALSE;
ELSE
	_Dequeue												:= FALSE;
END_IF
END_METHOD

METHOD PROTECTED _enqueue : BOOL //TRUE if method was successful
VAR_INPUT
	pData													: 	POINTER TO BYTE := 0;
	SizeOfData												: 	UDINT := 0;
	pMemory													: 	POINTER TO BYTE := 0;
	SizeOfMemory											: 	UDINT := 0;
END_VAR
IF pData = 0
	OR SizeOfData = 0
	OR pMemory = 0
	OR SizeOfMemory = 0
	OR Full AND NOT Overwrite
THEN
	_Enqueue												:= FALSE;
	RETURN;
ELSIF TestAndSet(Interlock)
THEN	
	_Enqueue												:= TRUE;
		
	(* maximum count *)
	MaxEntrys 												:= SizeOfMemory / SizeOfData;
	SizeOfEntry												:= SizeOfData;

	(* copy datasets *)
	MEMMOVE(pMemory + SizeOfData, pMemory, SEL(Full AND Overwrite,Count * SizeOfData , (Count - 1) * SizeOfData));
	
	(* copy datasets at the beginning *)
	MEMCPY(pMemory,pData,SizeOfData);
	Count													:= MIN(Count + 1, MaxEntrys);
	Empty 													:= FALSE;
	Full 													:= Count >= MaxEntrys;
	Interlock												:= FALSE;
ELSE
	_Enqueue												:= FALSE;
END_IF
END_METHOD

//Check wheter a value already exist
METHOD PROTECTED _isEnqueued : UDINT //data exist in Fifo if reurn value <> 0, returns index of entry in buffer 
VAR_INPUT
	pData													: 	POINTER TO BYTE := 0;
	SizeOfData												: 	UDINT := 0;
	pMemory													: 	POINTER TO BYTE := 0;
	SizeOfMemory											: 	UDINT := 0;
END_VAR	
VAR
	i 														: 	UDINT;
END_VAR
IF 	pData = 0
	OR SizeOfData = 0
	OR pMemory = 0
	OR SizeOfMemory = 0
	OR Empty
THEN
	_IsEnqueued												:= 0;
	RETURN;
ELSIF TestAndSet(Interlock)
THEN	
	_IsEnqueued												:= 0;
	MaxEntrys 												:= SizeOfMemory / SizeOfData;
	FOR i := 1 TO Count
	DO
		IF MEMCMP(pData,pMemory + ((i - 1) * SizeOfData), SizeOfData) = 0
		THEN
			_isEnqueued										:= i;
			EXIT;
		END_IF
	END_FOR
	Interlock												:= FALSE;
END_IF
END_METHOD

//Check wheter a value will be the next output of the buffer
METHOD PROTECTED _isNextEntry : BOOL //Inputs value is the next output 
VAR_INPUT
	pData													: 	POINTER TO BYTE := 0;
	SizeOfData												: 	UDINT := 0;
	pMemory													: 	POINTER TO BYTE := 0;
	SizeOfMemory											: 	UDINT := 0;
END_VAR
VAR
END_VAR
_IsNextEntry 	:= 0 = MEMCMP(pData,pMemory +(TO_UDINT(Count -1) * SizeOfData), SizeOfData) and NOT Empty;
END_METHOD

METHOD PROTECTED _readEntry : BOOL //TRUE if method was successful
VAR_INPUT
	idx														:	UDINT;
	pData													: 	POINTER TO BYTE := 0;
	SizeOfData												: 	UDINT := 0;
	pMemory													: 	POINTER TO BYTE := 0;
	SizeOfMemory											: 	UDINT := 0;
END_VAR
IF 	pData = 0
	OR SizeOfData = 0
	OR pMemory = 0
	OR SizeOfMemory = 0
	OR Empty
THEN
	_ReadEntry												:= FALSE;
	RETURN;
ELSIF TestAndSet(Interlock)
THEN	
	MaxEntrys 												:= SizeOfMemory / SizeOfData;
	IF idx < 1 OR idx > MIN(Count,MaxEntrys)
	THEN
		_ReadEntry											:= FALSE;
	ELSE
		MEMCPY(pData,pMemory + ((idx - 1) * SizeOfData), SizeOfData);
		_ReadEntry											:= TRUE;					
	END_IF
	Interlock												:= FALSE;
END_IF
END_METHOD

